// TwinCAT 3 PLC project Untitled1
// ProgramVersion: 3.1.4023.0
// libraries:
//   CmpBitmapPool, * (System)
//   Tc2_MC2, * (Beckhoff Automation GmbH)
//   Tc2_Standard, * (Beckhoff Automation GmbH)
//   Tc2_System, * (Beckhoff Automation GmbH)
//   Tc2_Utilities, * (Beckhoff Automation GmbH)
//   Tc3_Module, * (Beckhoff Automation GmbH)
//   Tc3_PackML_V2, * (Beckhoff Automation GmbH)
// project tree:
//   DUTs/ A21ToolStorage.TcDUT (not stored), Bundle.TcDUT (not stored), Interval.TcDUT (not stored), PositionMaterials.TcDUT (not stored)
//   DUTs/Alarms and Status/ A21Alarms.TcPOU, PMLStackLight.TcPOU (not stored)
//   DUTs/Enums/ A21.TcDUT (not stored), Chipboard.TcDUT (not stored), ConveyorMode.TcDUT (not stored), SectionEnum.TcDUT (not stored), Surface.TcDUT (not stored), WoodBunk.TcDUT (not stored)
//   DUTs/Insertion Package/Drives/ AirPiston.TcPOU (not stored), ClearLinkMC.TcPOU, SimplePiston.TcPOU
//   DUTs/Insertion Package/ Homing.TcDUT (not stored), Insertion.TcPOU, SuctionPad.TcDUT (not stored)
//   DUTs/Insertion Package/Prototypes/ FBA_Drive.TcPOU (not stored), FBA_TrifectaDrive.TcPOU, I_ContinuousDrive.TcIO (not stored), I_Drive.TcIO (not stored), I_EncodedDrive.TcIO (not stored), I_PositionalDrive.TcIO
//   DUTs/Machines/ Conveyor.TcPOU, ConveyorLL.TcPOU, EOAT.TcDUT (not stored), KukaRobot.TcPOU (not stored), RobotA21.TcPOU (not stored), StrapMachine.TcPOU (not stored)
//   DUTs/Material Holders/ MaterialHolder.TcPOU (not stored), MaterialSlot.TcDUT (not stored), SkidMagazine.TcPOU (not stored), StagingTable.TcPOU (not stored)
//   GVLs/ ContainerArrays.TcGVL (not stored), GVL.TcGVL (not stored), Hardware.TcGVL, Misc.TcGVL (not stored)
//   / PlcTask.TcTTO (not stored)
//   POUs/A21a - Chipboard/AOIs/ AOI_LoadChipboard.TcPOU (not stored)
//   POUs/A21b - Wood Bunk/AOIs/ AOI_LoadWoodBunk.TcPOU, AOI_StageWoodBunk.TcPOU (not stored), AOI_StagingTemplate.TcPOU
//   POUs/ CallHardware.TcPOU, FB_System.TcPOU, MAIN.TcPOU
//   POUs/Hardware Functions/ InsertionQuality.TcPOU (not stored), SetSuctionsPtrArr.TcPOU (not stored), SuctionQuality.TcPOU (not stored), SuctionQualityPtrArr.TcPOU (not stored), SetSuctions.TcPOU (not stored), SetupHardware.TcPOU (not stored)
//   POUs/A21a - Chipboard/ ChipboardEx.TcPOU
//   POUs/A21b - Wood Bunk/ WoodBunkEx.TcPOU
//   POUs/Utility/ AddToArray.TcPOU, AddToStringArray.TcPOU (not stored), ArrayIsEmpty.TcPOU, CleanStringsArray.TcPOU (not stored), IntegerBitAccess.TcPOU (not stored), IntegerToBoolArray.TcPOU (not stored), JoinStrings.TcPOU (not stored), WithinTolerance.TcPOU (not stored)
// real-time tasks:
//   TASK PlcTask: cycle T#10ms, priority 20, ADS port 350
// I/O:
//   DEVICE Device 1 (EtherCAT) (disabled), AmsNetId 192.168.101.188.2.1
//     EK1200 [EK1200-5000 EtherCAT Power supply (2A E-Bus)]
//       IPC_O [EL2809 16Ch. Dig. Output 24V, 0.5A]
//       JUNC_A21 [EK1122 2 port EtherCAT junction]
//         A21_C4 [EK1100 EtherCAT Coupler (2A E-Bus)]
//           A21_C4_I1 [EL1809 16Ch. Dig. Input 24V, 3ms]
//           A21_C4_O2 [EL2809 16Ch. Dig. Output 24V, 0.5A]
//           A21_C4_O3 [EL2809 16Ch. Dig. Output 24V, 0.5A]
//           BRIDGE_ROBOT1 [EL6695 EtherCAT Bridge terminal (Primary)]
//           A21_C4_END [EL9011 End Terminal]
//         A21_SB01 [EP1809-0021 16 Ch. Dig. Input 24V, 3ms, M8]
//         A21_SB05 [EP1008-0001 8 Ch. Dig. Input 24V, 3ms, M8]
//         A21_SB04 [EP1809-0021 16 Ch. Dig. Input 24V, 3ms, M8]
//         A21_SB03 [EP1008-0001 8 Ch. Dig. Input 24V, 3ms, M8]
//         A21_C1 [EK1100 EtherCAT Coupler (2A E-Bus)]
//           A21_C1_I1 [EL1809 16Ch. Dig. Input 24V, 3ms]
//           A21_C1_O2 [EL2809 16Ch. Dig. Output 24V, 0.5A]
//           BRIDGE_ROBOT2 [EL6695 EtherCAT Bridge terminal (Primary)]
//           A21_C1_END [EL9011 End Terminal]
//         A21_SB02 [EP1809-0021 16 Ch. Dig. Input 24V, 3ms, M8]
//         A21_SB07 [EP1008-0001 8 Ch. Dig. Input 24V, 3ms, M8]
//         A21_SB06 [EP1008-0001 8 Ch. Dig. Input 24V, 3ms, M8]
//   DEVICE Device 2 (TC3 EIP Scanner) (disabled), AmsNetId 192.168.101.188.3.1
//     ClearLink // <INFO> 169.254.0.152, ClearLink (ProdCode: 1, Rev: 2.93, Mac: 24:15:10:b0:30:37) </INFO> <EDS> C:\TwinCAT\3.1\Config\Io\EtherNetIP\clearlink_2.92.eds </EDS>
// variable links:
//   Untitled1/Untitled1 Instance <-> Device 1 (EtherCAT)/EK1200/JUNC_A21/A21_C1/A21_C1_I1
//     PlcTask Inputs/Hardware.strapperA21.atBundleLevel <-> Channel 6/Input
//     PlcTask Inputs/Hardware.strapperA21.done <-> Channel 4/Input
//     PlcTask Inputs/Hardware.strapperA21.error <-> Channel 1/Input
//     PlcTask Inputs/Hardware.strapperA21.home <-> Channel 5/Input
//     PlcTask Inputs/Hardware.strapperA21.ready <-> Channel 2/Input
//   Untitled1/Untitled1 Instance <-> Device 1 (EtherCAT)/EK1200/JUNC_A21/A21_C1/A21_C1_O2
//     PlcTask Outputs/Hardware.strapperA21.enable <-> Channel 2/Output
//     PlcTask Outputs/Hardware.strapperA21.execute <-> Channel 1/Output
//     PlcTask Outputs/Hardware.strapperA21.reset <-> Channel 3/Output
//   Untitled1/Untitled1 Instance <-> Device 1 (EtherCAT)/EK1200/JUNC_A21/A21_C1/BRIDGE_ROBOT2
//     PlcTask Inputs/Hardware.robot2.inputs[{2..20}] <-> IO Inputs/In_{2..20}  (19 links)
//     PlcTask Inputs/Hardware.robot2.inputs[1] <-> IO Inputs/In
//     PlcTask Inputs/Hardware.robot2.offline <-> SYNC Inputs/External device not connected
//     PlcTask Outputs/Hardware.robot2.outputs[{2..20}] <-> IO Outputs/Out_{2..20}  (19 links)
//     PlcTask Outputs/Hardware.robot2.outputs[1] <-> IO Outputs/Out
//   Untitled1/Untitled1 Instance <-> Device 1 (EtherCAT)/EK1200/JUNC_A21/A21_C4/A21_C4_I1
//     PlcTask Inputs/Hardware.suctionA21Top[1].occupied <-> Channel 9/Input
//     PlcTask Inputs/Hardware.suctionA21Top[2].occupied <-> Channel 10/Input
//     PlcTask Inputs/Hardware.suctionA21Top[3].occupied <-> Channel 11/Input
//     PlcTask Inputs/Hardware.verticalDriveA21Left.home <-> Channel 3/Input
//     PlcTask Inputs/Hardware.verticalDriveA21Left.innerLimit <-> Channel 1/Input
//     PlcTask Inputs/Hardware.verticalDriveA21Left.outerLimit <-> Channel 2/Input
//     PlcTask Inputs/Hardware.verticalDriveA21Right.home <-> Channel 7/Input
//     PlcTask Inputs/Hardware.verticalDriveA21Right.innerLimit <-> Channel 5/Input
//     PlcTask Inputs/Hardware.verticalDriveA21Right.outerLimit <-> Channel 6/Input
//   Untitled1/Untitled1 Instance <-> Device 1 (EtherCAT)/EK1200/JUNC_A21/A21_C4/A21_C4_O2
//     PlcTask Outputs/Hardware.horizontalDriveA21Left.valveExtend <-> Channel 5/Output
//     PlcTask Outputs/Hardware.horizontalDriveA21Left.valveRetract <-> Channel 6/Output
//     PlcTask Outputs/Hardware.horizontalDriveA21Right.valveExtend <-> Channel 15/Output
//     PlcTask Outputs/Hardware.horizontalDriveA21Right.valveRetract <-> Channel 16/Output
//     PlcTask Outputs/Hardware.suctionA21Left[{1..4}].enable <-> Channel {7..10}/Output  (4 links)
//     PlcTask Outputs/Hardware.verticalDriveA21Left.brakeRelease <-> Channel 4/Output
//     PlcTask Outputs/Hardware.verticalDriveA21Right.brakeRelease <-> Channel 14/Output
//   Untitled1/Untitled1 Instance <-> Device 1 (EtherCAT)/EK1200/JUNC_A21/A21_C4/A21_C4_O3
//     PlcTask Outputs/Hardware.pistonA21Bottom.pistonExtend <-> Channel 5/Output
//     PlcTask Outputs/Hardware.pistonA21Bottom.pistonRetract <-> Channel 6/Output
//     PlcTask Outputs/Hardware.suctionA21Bottom[1].enable <-> Channel 7/Output
//     PlcTask Outputs/Hardware.suctionA21Bottom[2].enable <-> Channel 8/Output
//     PlcTask Outputs/Hardware.suctionA21Right[{1..4}].enable <-> Channel {1..4}/Output  (4 links)
//     PlcTask Outputs/Hardware.suctionA21Top[1].enable <-> Channel 9/Output
//     PlcTask Outputs/Hardware.suctionA21Top[2].enable <-> Channel 10/Output
//     PlcTask Outputs/Hardware.suctionA21Top[3].enable <-> Channel 11/Output
//   Untitled1/Untitled1 Instance <-> Device 1 (EtherCAT)/EK1200/JUNC_A21/A21_C4/BRIDGE_ROBOT1
//     PlcTask Inputs/Hardware.robot1.inputs[{2..20}] <-> IO Inputs/In_{2..20}  (19 links)
//     PlcTask Inputs/Hardware.robot1.inputs[1] <-> IO Inputs/In
//     PlcTask Inputs/Hardware.robot1.offline <-> SYNC Inputs/External device not connected
//     PlcTask Outputs/Hardware.robot1.outputs[{2..20}] <-> IO Outputs/Out_{2..20}  (19 links)
//     PlcTask Outputs/Hardware.robot1.outputs[1] <-> IO Outputs/Out
//   Untitled1/Untitled1 Instance <-> Device 1 (EtherCAT)/EK1200/JUNC_A21/A21_SB01
//     PlcTask Inputs/ContainerArrays.tableHmiA21Left[{1..10}].occupied <-> Channel {1..10}/Input  (10 links)
//     PlcTask Inputs/Hardware.horizontalDriveA21Left.home <-> Channel 11/Input
//     PlcTask Inputs/Hardware.insertionA21Left.contact <-> Channel 12/Input
//     PlcTask Inputs/Hardware.suctionA21Left[{1..4}].occupied <-> Channel {13..16}/Input  (4 links)
//   Untitled1/Untitled1 Instance <-> Device 1 (EtherCAT)/EK1200/JUNC_A21/A21_SB02
//     PlcTask Inputs/ContainerArrays.tableHmiA21Right[{1..10}].occupied <-> Channel {1..10}/Input  (10 links)
//     PlcTask Inputs/Hardware.horizontalDriveA21Right.home <-> Channel 11/Input
//     PlcTask Inputs/Hardware.insertionA21Right.contact <-> Channel 12/Input
//     PlcTask Inputs/Hardware.suctionA21Right[{1..4}].occupied <-> Channel {13..16}/Input  (4 links)
//   Untitled1/Untitled1 Instance <-> Device 1 (EtherCAT)/EK1200/JUNC_A21/A21_SB07
//     PlcTask Inputs/Hardware.pistonA21Bottom.extended <-> Channel 5/Input
//     PlcTask Inputs/Hardware.pistonA21Bottom.retracted <-> Channel 4/Input
//     PlcTask Inputs/Hardware.suctionA21Bottom[1].occupied <-> Channel 6/Input
//     PlcTask Inputs/Hardware.suctionA21Bottom[2].occupied <-> Channel 7/Input
//   Untitled1/Untitled1 Instance <-> Device 2 (TC3 EIP Scanner)/ClearLink
//     PlcTask Inputs/Hardware.verticalDriveA21Left.hlfb <-> Connection 1 (Input/Output)/Inputs/Motor0 HLFB Duty
//     PlcTask Inputs/Hardware.verticalDriveA21Right.hlfb <-> Connection 1 (Input/Output)/Inputs/Motor1 HLFB Duty
//     PlcTask Outputs/Hardware.verticalDriveA21Left.outputRegister <-> Connection 1 (Input/Output)/Outputs/Motor0 Out Reg
//     PlcTask Outputs/Hardware.verticalDriveA21Left.pulse <-> Connection 1 (Input/Output)/Outputs/Motor0 Trig Pulses
//     PlcTask Outputs/Hardware.verticalDriveA21Right.outputRegister <-> Connection 1 (Input/Output)/Outputs/Motor1 Out Reg
//     PlcTask Outputs/Hardware.verticalDriveA21Right.pulse <-> Connection 1 (Input/Output)/Outputs/Motor1 Trig Pulses

// ---- GVLs/Hardware.TcGVL
//{attribute 'qualified_only'}
VAR_GLOBAL
	robot1 : RobotA21;
	robot2 : RobotA21;
	
	toolStorageA21Left : A21ToolStorage;
	toolStorageA21Right : A21ToolStorage;
	
	skidA21Left : SkidMagazine;
	skidA21Right : SkidMagazine;
	
	magazineA21Left : SkidMagazine;
	magazineA21Right : SkidMagazine;
	stagingTableLeft : StagingTable;
	stagingTableRight : StagingTable;
	
	strapperA21 : StrapMachine;
	
	horizontalDriveA21Left, horizontalDriveA21Right : AirPiston := (
		limitSensorDefaultState := FALSE,
		useBrake := FALSE);
	
	verticalDriveA21Left, verticalDriveA21Right : ClearLinkMC := (
		limitSensorDefaultState := TRUE, 
		homingDirectionOut := TRUE, //outwards (up)
		minPosition := 0,
		displacementPerRotation := 1,
		unitsPerPulse := 8000); //0.1x gearbox, 10 revs/pulse to compensate
		
	insertionA21Left, insertionA21Right : Insertion;
	
	pistonA21Bottom : SimplePiston;
	
	suctionA21Top : ARRAY[1..3] OF SuctionPad;
	suctionA21Left : ARRAY[1..4] OF SuctionPad;
	suctionA21Right : ARRAY[1..4] OF SuctionPad; 
	suctionA21Bottom : ARRAY[1..2] OF SuctionPad;
	
	stackLightA21 : PMLStackLight;
	alarmsA21 : A21Alarms;
END_VAR

// ---- DUTs/Insertion Package/Prototypes/I_PositionalDrive.TcIO
INTERFACE I_PositionalDrive EXTENDS I_Drive

PROPERTY CurrentPosition : LREAL
GET
END_GET
SET
END_SET
END_PROPERTY

METHOD ABSTRACT moveAbsolute : BOOL
VAR_INPUT
	newTarget : LREAL; 
END_VAR
END_METHOD

METHOD ABSTRACT moveRelative : BOOL
VAR_INPUT
	distance : LREAL;
END_VAR
END_METHOD

PROPERTY TargetPosition : LREAL
GET
END_GET
SET
END_SET
END_PROPERTY

END_INTERFACE

// ---- DUTs/Insertion Package/Drives/ClearLinkMC.TcPOU
FUNCTION_BLOCK ClearLinkMC EXTENDS FBA_TrifectaDrive IMPLEMENTS I_EncodedDrive
VAR_OUTPUT
	pulse AT %Q* : INT;
	brakeRelease AT %Q* : BOOL := TRUE;
	enable : BOOL;
	A : BOOL;
	B : BOOL;
	clear : BOOL;
END_VAR
VAR	
	hlfb AT %I* : REAL := -9999; //high level feedback, if -9999 then servo is idle
	
	outputRegister AT %Q* : INT;
	pulseRequest : INT;
	
	homingDelay : TON;
	resetPulse : TP;
	
	mode : (HOLD, TARGET, CONTINUOUS, RESET_ERR);
	calculation : (IDLE, DOWN, UP, CALCULATE, DONE);
	maxPosition : LREAL;
	
	position, targetPos : LREAL;
	
	pulsePosition : INT;
	pulseCounter : INT;
	rotationsPerPulse : INT; //revolutions per pulse
	displacementPerPulse : LREAL; //displacement per pulse
END_VAR
VAR_STAT CONSTANT
	resetWidth : TIME := T#500MS;
	delayWidth : TIME := T#500MS;
END_VAR
VAR //constructor
	homingDirectionOut : BOOL; 			//homing direction - see <A>
	minPosition : LREAL;
	displacementPerRotation : LREAL; 	//displacement per revolution	
	unitsPerPulse : INT := 800; 		//800 Teknic units per rotation - default setting is 800 units (1 rotation) per pulse
END_VAR

//M-connector output register
outputRegister.0 := enable AND bEnable; 	//enable
outputRegister.1 := A; 						//direction bit - T = outwards, F = inwards
outputRegister.2 := B; 						//homing bit - after startup, set to TRUE to begin homing, then set to FALSE to finish homing
outputRegister.3 := clear; 					//reset bit

rotationsPerPulse := unitsPerPulse/800; //Teknic constant - 800 units per rotation
displacementPerPulse := displacementPerRotation * rotationsPerPulse;

resetPulse(IN:= , PT:= resetWidth, Q=> clear, ET=> ); //reset pulse

IF NOT enable AND NOT AtInnerLimit THEN
	homingComplete := FALSE;
	step := Homing.IDLE;
	mode := HOLD;
END_IF

override();

CASE mode OF		
	HOLD: //hold current position, no motion
		pulse := 0;
		pulseRequest := 0;
	
	TARGET:	//target a given position
		
		IF WithinTolerance(position, targetPos, displacementPerPulse) THEN
			pulseRequest := 0;
			pulse := 0;
			mode := HOLD;
			
		ELSIF NOT Active THEN
			A :=  position < targetPos;
			(*
			2 options to traverse to a target position:
				a)  send all pulses at once - continuous motion but may exceed limits, check for bounds before setting
				b)  1 pulse at a time - choppy but safer
			*)
			targetPos := MAX(targetPos, minPosition); //if below minPosition, set to minPosition
			targetPos := MIN(targetPos, maxPosition); //if above maxPosition, set to maxPosition
			
			pulseRequest := TO_INT(ABS(position - targetPos)/displacementPerPulse);
			//pulseRequest := 1;
		END_IF
		
	CONTINUOUS: //single pulses in the direction specified by moveContinuous()
		pulseRequest := 1;
		
	RESET_ERR: //reset pulse, servo may need to be rehomed aftewards
		pulse := 0;
		pulseRequest := 0;
		resetPulse.IN := TRUE;
		
		IF resetPulse.Q THEN
			resetPulse.IN := FALSE;
			mode := HOLD;
		END_IF
		
END_CASE

sequence();

PROPERTY Active : BOOL
GET
Active := hlfb <> -9999;
END_GET
END_PROPERTY

{attribute 'monitoring':='call'}
PROPERTY AtOuterLimit : BOOL
GET
AtOuterLimit := outerLimit <> limitSensorDefaultState;
END_GET
END_PROPERTY

METHOD PRIVATE calculatePositions : BOOL
(*
the purpose of this method is calculate the position at the outer limit

complete a full range traverse while counting the pulses, then multiply
	displacement per rotation
	rotations per pulse
	number of pulses for the traversal
and add to position at inner limit to get position at outer limit
*)
CASE calculation OF
	IDLE:
		calculation := DOWN;
		
	DOWN:
		moveContinuous(direction := MC_Negative_Direction);
		IF AtInnerLimit THEN
			calculation := UP;
			pulseCounter := 0;
		END_IF
		
	UP:
		moveContinuous(direction := MC_Positive_Direction);
		IF AtHome THEN
			maxPosition := minPosition + (displacementPerRotation * rotationsPerPulse * pulseCounter);
			calculation := DONE;
		END_IF
		
	DONE:
		calculation := 0;
		calculatePositions := TRUE;
		
END_CASE
END_METHOD

PROPERTY CurrentPosition : LREAL
GET
CurrentPosition := position;

//CurrentPosition := pulsePosition * displacementPerPulse;
END_GET
SET
position := CurrentPosition;
END_SET
END_PROPERTY

PROPERTY Error : BOOL
GET
END_GET
END_PROPERTY

METHOD homingSequence : BOOL
homingDelay(IN:= , PT:= delayWidth, Q=> , ET=> );

CASE step OF
	Homing.IDLE:
		enable := TRUE;
		A := FALSE;
		B := TRUE;
		brakeRelease := TRUE;
		
		homingComplete := FALSE;
		
		homingDelay.IN := TRUE;
		IF homingDelay.Q THEN
			homingDelay.IN := FALSE;
			//step := Homing.START;
			step := Homing.RETRY;
		END_IF
		
	Homing.START:
		IF homingDelay.Q THEN
			homingDelay.IN := FALSE;
			step := Homing.SET;
			
		ELSIF AtHome THEN
			homingDelay.IN := TRUE;
			
		ELSIF AtOuterLimit THEN
			step := Homing.RETRY;
		
		ELSE
			enable := TRUE;
			A := FALSE;
			B := TRUE;
			brakeRelease := TRUE;
		
		END_IF
	
	Homing.RETRY:
		IF AtInnerLimit THEN
			homingDelay.IN := TRUE;
			enable := FALSE;
			
			IF homingDelay.Q THEN
				homingDelay.IN := FALSE;
				step := Homing.START;
			END_IF
			
		ELSE
			enable := TRUE;
			A := FALSE;
			B := FALSE;
			brakeRelease := TRUE;
			
			mode := CONTINUOUS;
		END_IF

	Homing.SET:
		enable := TRUE;
		A := FALSE;
		B := FALSE;
		brakeRelease := TRUE;
		
		IF calculatePositions() THEN
			step := Homing.DONE;
		END_IF
		
	Homing.DONE:
		homingSequence := homingComplete := TRUE;
		
		pulsePosition := 0;
		
		mode := HOLD;
		step := Homing.IDLE;
	
END_CASE
END_METHOD

{attribute 'TcRpcEnable'}
METHOD moveAbsolute : BOOL
VAR_INPUT
	newTarget : LREAL;
END_VAR
IF target >= maxPosition AND target <= minPosition THEN
	A :=  position < targetPos;
	targetPos := newTarget;
	mode := TARGET;
	
	moveAbsolute := TRUE;
END_IF
END_METHOD

{attribute 'TcRpcEnable'}
METHOD moveContinuous : BOOL
VAR_INPUT
	direction : MC_Direction;
END_VAR
IF direction = MC_Negative_Direction THEN
	A := FALSE;
ELSIF direction = MC_Positive_Direction THEN
	A := TRUE;
END_IF

mode := CONTINUOUS;
END_METHOD

{attribute 'TcRpcEnable'}
METHOD moveRelative : BOOL
VAR_INPUT
	distance : LREAL;
END_VAR
targetPos := targetPos + distance;

mode := TARGET;
END_METHOD

METHOD PRIVATE override : BOOL
VAR_INPUT
END_VAR
(*
allowable motion is between AtHome and AtInnerLimit
*)
IF AtHome AND NOT Active THEN
	IF homingDirectionOut THEN //homing is outwards
		position := maxPosition;
		pulsePosition := pulseCounter;
	ELSE
		position := minPosition;
		pulsePosition := 0;
	END_IF
	

ELSIF AtInnerLimit AND NOT Active THEN
	IF homingDirectionOut THEN //homing is outwards
		position := minPosition;
		pulsePosition := 0;
	ELSE
		position := maxPosition;
		pulsePosition := pulseCounter;
	END_IF
END_IF

CASE mode OF		
	HOLD:
		//
	
	TARGET:
		IF
			(AtHome AND TargetPosition > CurrentPosition) OR
			(AtInnerLimit AND TargetPosition > CurrentPosition) OR
			(AtOuterLimit AND TargetPosition < CurrentPosition)
		THEN
			mode := HOLD;
		END_IF
		
	CONTINUOUS:
		IF
			(AtHome AND A) OR
			(AtInnerLimit AND A) OR
			(AtOuterLimit AND NOT A)
		THEN
			mode := HOLD;
		END_IF
		
	RESET_ERR:
		//
		
END_CASE
END_METHOD

METHOD reset : BOOL
VAR_INPUT
END_VAR
mode := RESET_ERR;
END_METHOD

METHOD PRIVATE sequence : BOOL
VAR_INPUT
END_VAR
IF Active THEN //servo is active
	IF A THEN //positive direction
		position := position + (displacementPerPulse * pulse);
		pulsePosition := pulsePosition + pulse;
		
		pulseCounter := pulseCounter + pulse;
	ELSE //negative direction
		position := position - (displacementPerPulse * pulse);
		pulsePosition := pulsePosition - pulse;
		
		pulseCounter := pulseCounter - pulse;
	END_IF
	pulse := 0; //pulses already received, can be set to 0 so position change is not compounded

ELSIF pulse = 0 THEN //servo is not active
	pulse := pulseRequest;
END_IF

pulseRequest := 0; //remove this if not working as intended
END_METHOD

METHOD stop : BOOL
VAR_INPUT
END_VAR
mode := HOLD;
END_METHOD

PROPERTY TargetPosition : LREAL
GET
END_GET
SET
targetPos := TargetPosition;
END_SET
END_PROPERTY

METHOD toHome : BOOL
VAR_INPUT
END_VAR
IF homingDirectionOut THEN
	moveAbsolute(newTarget := maxPosition);
ELSE
	moveAbsolute(newTarget := minPosition);
END_IF
END_METHOD

END_FUNCTION_BLOCK

// ---- DUTs/Insertion Package/Prototypes/FBA_TrifectaDrive.TcPOU
FUNCTION_BLOCK ABSTRACT FBA_TrifectaDrive EXTENDS FBA_Drive
VAR
	outerLimit AT %I* : BOOL;
END_VAR
(*
this abstract FB adds a rear limit sensor to FBA_Drive
*)

{attribute 'monitoring':='call'}
PROPERTY AtOuterLimit : BOOL
GET
AtOuterLimit := outerLimit <> limitSensorDefaultState;
END_GET
END_PROPERTY

END_FUNCTION_BLOCK

// ---- DUTs/Insertion Package/Insertion.TcPOU
FUNCTION_BLOCK Insertion //2d insertion that combines a slider (alignment) and screw (push)
VAR_INPUT
	enable : BOOL;
END_VAR
VAR_INPUT //interface references to existing drives
	slider : I_EncodedDrive;
	screw : I_ContinuousDrive;
END_VAR
VAR_OUTPUT
	contact AT %I* : BOOL;
	
	active : BOOL;
	error : BOOL;
	home : BOOL;
	
	homingComplete : BOOL;
	
	sliderPos : LREAL;
END_VAR
(*
this FB encapsulates 2 drives into a generic insertion machine
both drives should be declared externally in Hardware GVL as a concrete FB
Insertion instance should be declared and called in module scope, with the drives from Hardware GVL passed in by Interface reference
*)

homingComplete := slider.HomeSet AND screw.HomeSet;

active := slider.Active OR screw.Active;
error := slider.Error OR screw.Error;
home := slider.AtHome AND screw.AtHome;

sliderPos := slider.CurrentPosition;

METHOD align : BOOL
VAR_INPUT
	targetPos : REAL;
END_VAR
slider.moveAbsolute(newTarget := targetPos);
END_METHOD

METHOD homingSequence : BOOL
VAR_INPUT
END_VAR
IF NOT slider.homeSet THEN
	slider.homingSequence();
END_IF

IF NOT screw.homeSet THEN
	screw.homingSequence();
END_IF

homingSequence := homingComplete;
END_METHOD

METHOD press : BOOL
VAR_INPUT
END_VAR
screw.moveContinuous(direction := MC_Negative_Direction);
END_METHOD

METHOD release : BOOL
VAR_INPUT
END_VAR
screw.moveContinuous(direction := MC_Positive_Direction);
END_METHOD

METHOD reset : BOOL
VAR_INPUT
END_VAR
slider.reset();
screw.reset();
END_METHOD

METHOD stop : BOOL
VAR_INPUT
END_VAR
screw.stop();
slider.stop();
END_METHOD

METHOD toHome : BOOL
VAR_INPUT
END_VAR
slider.toHome();
screw.toHome();

toHome := slider.AtHome AND screw.AtHome;
END_METHOD

METHOD traverse : BOOL
VAR_INPUT
	direction : MC_Direction;
END_VAR
slider.moveContinuous(direction := MC_Negative_Direction);
END_METHOD

END_FUNCTION_BLOCK

// ---- DUTs/Insertion Package/Drives/SimplePiston.TcPOU
FUNCTION_BLOCK SimplePiston
VAR_INPUT
	bEnable : BOOL;
END_VAR
VAR_OUTPUT
	pistonExtend AT %Q* : BOOL;
	pistonRetract AT %Q* : BOOL;
	
	extended AT %I* : BOOL;
	retracted AT %I* : BOOL;
	
	busy : BOOL;
END_VAR
VAR
	mode : (HOLD, IN, OUT);
END_VAR

IF
	NOT bEnable OR
	(retracted AND_THEN (pistonRetract OR mode = OUT)) OR
	(extended AND_THEN (pistonExtend OR mode = IN))
THEN
	mode := HOLD;
END_IF

CASE mode OF
	HOLD:
		pistonRetract := FALSE;
		pistonExtend := FALSE;
		
	IN:
		pistonRetract := FALSE;
		pistonExtend := TRUE;
	
	OUT:
		pistonRetract := TRUE;
		pistonExtend := FALSE;
	
END_CASE

busy := mode = IN OR mode = OUT;

METHOD extend : BOOL
VAR_INPUT
END_VAR
mode := IN;
END_METHOD

METHOD retract : BOOL
VAR_INPUT
END_VAR
mode := OUT;

retract := retracted;
END_METHOD

METHOD stop : BOOL
VAR_INPUT
END_VAR
pistonExtend := FALSE;
pistonRetract := FALSE;
mode := HOLD;
END_METHOD

END_FUNCTION_BLOCK

// ---- DUTs/Alarms and Status/A21Alarms.TcPOU
FUNCTION_BLOCK A21Alarms
VAR_OUTPUT
	panelPowerOn : BOOL;
	safetyOk : BOOL;
	airPressureOk : BOOL;
END_VAR
VAR_OUTPUT
	alarm : BOOL;
END_VAR

alarm :=
	NOT panelPowerOn OR 
	NOT safetyOk OR
	NOT airPressureOk;

END_FUNCTION_BLOCK

// ---- DUTs/Machines/Conveyor.TcPOU
FUNCTION_BLOCK Conveyor
VAR
	enable AT %Q* : BOOL := TRUE;
	direction AT %Q* : BOOL; //FALSE = forward, TRUE = backward
	pulse AT %Q* : BOOL;
	reset AT %Q* : BOOL;
	
	sensorEntry AT %I* : BOOL;
	sensorExit AT %I* : BOOL;

	lifterEnable AT %Q* : BOOL := TRUE;
	lifterDirection AT %Q* : BOOL; //FALSE = up, TRUE = down
	lifterPulse AT %Q* : BOOL;
	lifterReset AT %Q* : BOOL;
END_VAR
VAR_OUTPUT
	operation : ConveyorMode;
	request : ConveyorMode;
	
	error AT %I* : BOOL;
	lifterError AT %I* : BOOL;
	
	position AT %I* : REAL;
	velocity AT %I* : REAL;
	
	hasLifter : BOOL;
	extended AT %I* : BOOL;
	retracted AT %I* : BOOL;
END_VAR
VAR
	lifterMode : (HOLD, UP, DOWN); 
	lifterMode2 : (LIFTER_EXTEND, LIFTER_RETRACT);
	
	//pulses are assumed to be low-high-low
	pulser : TP;
	lifterPulser : TP;
END_VAR
VAR_STAT CONSTANT
	pulseWidth : TIME := T#25MS;
END_VAR
(*
this version of Conveyor is to be implemented as a linked list,
	allowing it to control its own mode internally -
	without the use of an external conveyor control module - 
	eliminating the ability for other modules to modify its mode
*)

lifterPulser(IN:= , PT:= pulseWidth, Q=> lifterPulse, ET=> );
lifterPulser.IN := 
	hasLifter AND
	lifterEnable AND 
	NOT lifterError AND 
	NOT lifterReset AND 
	( (lifterMode = LIFTER_EXTEND AND NOT extended) OR (lifterMode = LIFTER_RETRACT AND NOT retracted) ) AND
	lifterPulser.Q; //self-ending pulse

override();

CASE lifterMode OF
	HOLD:
		lifterDirection := TRUE;
		lifterPulse := FALSE;
		
	UP:
		lifterDirection := FALSE;
		lifterPulse := NOT lifterPulse;
	
	DOWN:
		lifterDirection := TRUE;
		lifterPulse := NOT lifterPulse;
	
END_CASE

//conveyors do not move independently like motion drives, their operation is set by an additional conveyor control module
traverseSequence();

METHOD backward : BOOL
VAR_INPUT
END_VAR
END_METHOD

METHOD extend : BOOL
VAR_INPUT
END_VAR
VAR
	noLifter : BOOL;
END_VAR
IF hasLifter THEN
	lifterMode := UP;
	extend := TRUE;
ELSE
	noLifter := TRUE;
END_IF
END_METHOD

METHOD forward : BOOL
VAR_INPUT
END_VAR
END_METHOD

METHOD occupied : BOOL
occupied := sensorExit OR sensorEntry;
END_METHOD

METHOD PRIVATE override : BOOL
VAR_INPUT
END_VAR
IF
	(extended AND lifterMode = UP) OR
	(retracted AND lifterMode = DOWN)
THEN
	lifterMode := HOLD;
END_IF
END_METHOD

METHOD reset : BOOL
VAR_INPUT
END_VAR
position := 0;
velocity := velocity; //no change

extend();
END_METHOD

METHOD retract : BOOL
VAR_INPUT
END_VAR
VAR
	noLifter : BOOL;
END_VAR
IF hasLifter THEN
	lifterMode := DOWN;
	retract := TRUE;
ELSE
	noLifter := TRUE;
END_IF
END_METHOD

METHOD setOperation : BOOL
VAR_INPUT
	newOperation : ConveyorMode;
END_VAR
operation := newOperation;
END_METHOD

METHOD setRequest : BOOL
VAR_INPUT
	requestedMode : ConveyorMode;
END_VAR
request := requestedMode;
END_METHOD

METHOD target : BOOL
VAR_INPUT
	targetPosition : REAL;
END_VAR
END_METHOD

METHOD PRIVATE traverseSequence : BOOL
VAR_INPUT
END_VAR
direction := (operation = ConveyorMode.BACKWARD);

pulser(IN:= , PT:= pulseWidth, Q=> pulse, ET=> );
pulser.IN := 
	enable AND 
	NOT error AND 
	NOT reset AND 
	(operation = ConveyorMode.FORWARD OR operation = ConveyorMode.BACKWARD)
	AND pulser.Q; //ends pulse itself
END_METHOD

END_FUNCTION_BLOCK

// ---- DUTs/Machines/ConveyorLL.TcPOU
FUNCTION_BLOCK ConveyorLL
VAR
	enable AT %Q* : BOOL := TRUE;
	direction AT %Q* : BOOL; //FALSE = forward, TRUE = backward
	pulse AT %Q* : BOOL;
	reset AT %Q* : BOOL;
	
	sensorEntry AT %I* : BOOL;
	sensorExit AT %I* : BOOL;

	lifterEnable AT %Q* : BOOL := TRUE;
	lifterDirection AT %Q* : BOOL; //FALSE = up, TRUE = down
	lifterPulse AT %Q* : BOOL;
	lifterReset AT %Q* : BOOL;
END_VAR
VAR_OUTPUT
	operation : ConveyorMode;
	request : ConveyorMode;
	
	error AT %I* : BOOL;
	lifterError AT %I* : BOOL;
	
	position AT %I* : REAL;
	velocity AT %I* : REAL;
	
	hasLifter : BOOL;
	extended AT %I* : BOOL;
	retracted AT %I* : BOOL;
END_VAR
VAR
	nextConveyor : POINTER TO Conveyor;
	prevConveyor : POINTER TO Conveyor;
	
	lifterMode : (HOLD, LIFTER_EXTEND, LIFTER_RETRACT); 
	
	//pulses are assumed to be low-high-low
	pulser : TP;
	lifterPulser : TP;
END_VAR
VAR_STAT CONSTANT
	pulseWidth : TIME := T#25MS;
END_VAR

pulser(IN:= , PT:= pulseWidth, Q=> pulse, ET=> );
pulser.IN := 
	enable AND 
	NOT error AND 
	NOT reset AND 
	(operation = ConveyorMode.FORWARD OR operation = ConveyorMode.BACKWARD)
	AND pulser.Q; //ends pulse itself

lifterPulser(IN:= , PT:= pulseWidth, Q=> lifterPulse, ET=> );
lifterPulser.IN := 
	hasLifter AND
	lifterEnable AND 
	NOT lifterError AND 
	NOT lifterReset AND 
	( (lifterMode = LIFTER_EXTEND AND NOT extended) OR (lifterMode = LIFTER_RETRACT AND NOT retracted) ) AND
	lifterPulser.Q; //self-ending pulse

override();

CASE lifterMode OF
	HOLD:
		lifterDirection := TRUE;
		lifterPulse := FALSE;
		
	LIFTER_EXTEND:
		lifterDirection := FALSE;
		lifterPulse := NOT lifterPulse;
	
	LIFTER_RETRACT:
		lifterDirection := TRUE;
		lifterPulse := NOT lifterPulse;
	
END_CASE

sequence();

METHOD backward : BOOL
VAR_INPUT
END_VAR
END_METHOD

METHOD extend : BOOL
VAR_INPUT
END_VAR
VAR
	noLifter : BOOL;
END_VAR
IF hasLifter THEN
	lifterMode := UP;
	extend := TRUE;
ELSE
	noLifter := TRUE;
END_IF
END_METHOD

METHOD forward : BOOL
VAR_INPUT
END_VAR
END_METHOD

PROPERTY IsOccupied : BOOL
GET
IsOccupied := sensorExit OR sensorEntry;
END_GET
END_PROPERTY

METHOD PRIVATE override : BOOL
VAR_INPUT
END_VAR
IF
	(extended AND lifterMode = UP) OR
	(retracted AND lifterMode = DOWN)
THEN
	lifterMode := HOLD;
END_IF
END_METHOD

METHOD reset : BOOL
VAR_INPUT
END_VAR
position := 0;
velocity := velocity; //no change

extend();
END_METHOD

METHOD retract : BOOL
VAR_INPUT
END_VAR
VAR
	noLifter : BOOL;
END_VAR
IF hasLifter THEN
	lifterMode := DOWN;
	retract := TRUE;
ELSE
	noLifter := TRUE;
END_IF
END_METHOD

METHOD PRIVATE sequence : BOOL
VAR_INPUT
END_VAR
VAR
	nextOp, prevOp : ConveyorMode;
END_VAR
IF nextConveyor <> 0 THEN
	nextOp := nextConveyor^.operation;
END_IF
IF prevConveyor <> 0 THEN
	prevOp := prevConveyor^.operation;
END_IF


IF IsOccupied THEN
	operation := MAX(nextOp, request, prevOp);
ELSE
	operation := ConveyorMode.IDLE;
END_IF


direction := (operation = ConveyorMode.BACKWARD); //set direction bit

IF hasLifter THEN
	
END_IF
END_METHOD

METHOD setOperation : BOOL
VAR_INPUT
	newOperation : ConveyorMode;
END_VAR
operation := newOperation;
END_METHOD

METHOD setRequest : BOOL
VAR_INPUT
	requestedMode : ConveyorMode;
END_VAR
request := requestedMode;
END_METHOD

METHOD target : BOOL
VAR_INPUT
	targetPosition : REAL;
END_VAR
END_METHOD

END_FUNCTION_BLOCK

// ---- POUs/A21b - Wood Bunk/AOIs/AOI_LoadWoodBunk.TcPOU
FUNCTION_BLOCK AOI_LoadWoodBunk
VAR_INPUT
	execute : BOOL;
END_VAR
VAR_IN_OUT CONSTANT
	sectionID : SectionEnum;
END_VAR
VAR_IN_OUT
	robot : RobotA21;
	table : StagingTable;
	//suctions : ARRAY[*] OF SuctionPad;
	//if assigned using . operator instead of (), this becomes a pointer - use numPads isntead of UPPER_BOUND/LOWER_BOUND
	loadedMaterials : ARRAY[*] OF STRING;
END_VAR
VAR_INPUT
	suctions : POINTER TO SuctionPad;
	surfaceID : Surface;
	material : STRING;	
	numPads : DINT;
END_VAR
VAR_OUTPUT
	busy : BOOL;
	done : BOOL;
	error : BOOL;
	
	recovery : BOOL;
	failCounter : INT;
	
	donePulse : BOOL;
END_VAR
VAR
	run : BOOL;
	trigger : R_TRIG;
	doneTrigger : R_TRIG;
	
	slot : INT;
	
	suctionTimer : TON;
	step : (IDLE, PREP_ROBOT, GET_FROM_TABLE, LOAD_TO_INSERTION, COMPLETE, RECOVERY_IDLE, RECOVERY_REMOVE, RECOVERY_STAGE);
END_VAR
VAR
	i : DINT;
	test : BOOL;
	
	iWoodBunk : WoodBunk;
END_VAR
VAR CONSTANT
	suctionDelay : TIME := T#2S;
	suctionDistance : INT := 10;
END_VAR

{warning disable C0371}

trigger(CLK:= execute, Q=> );
doneTrigger(CLK:= done, Q=> donePulse);
busy := trigger.Q OR step > 0;

IF step > IDLE AND_THEN NOT preExecution() THEN //conditions to track before execution
	RETURN;
END_IF

(*
if required bunk was not found on table - restage entire table
if bunk was not loaded correctly - remove bunk, then restage entire table
*)

CASE step OF
	IDLE:
		IF trigger.Q THEN //reset outputs
			done := FALSE;
			error := FALSE;
			recovery := FALSE;
			
			step := PREP_ROBOT;
		END_IF
		
	PREP_ROBOT:
		robot.clearCommand();
		IF robot.Ready THEN
			step := GET_FROM_TABLE;
			slot := 0;
		END_IF
		
	GET_FROM_TABLE:		
		IF slot < 1 AND_THEN NOT table.findSlot(material := material, index => slot) THEN
			step := RECOVERY_STAGE;
			RETURN;
		END_IF
		
		
		
		IF NOT table.isOccupied(i := slot) AND table.getSlot(i := slot) <> '' THEN //move from table to robot gripper
			robot.HoldMaterial := table.getSlot(i := slot);
			table.remove(i := slot, material => );
		END_IF
		
		IF robot.Done THEN
			step := COMPLETE;
			RETURN;
		ELSIF robot.materialAtHoldingPosition >= 1 AND robot.materialAtHoldingPosition <= 8 THEN
			step := LOAD_TO_INSERTION;
			RETURN;
		END_IF
		
		CASE surfaceID OF
			Surface.TOP: 					robot.setGroup(group := 1, value := A21.LOAD_BUNK_TOP); 
			Surface.LEFT, Surface.RIGHT: 	robot.setGroup(group := 1, value := A21.LOAD_BUNK_SIDE);
			Surface.BOTTOM: 				robot.setGroup(group := 1, value := A21.LOAD_BUNK_BOTTOM);
		END_CASE
		robot.setGroup(group := 2, value := slot); 
		
		FOR iWoodBunk:=0 TO WoodBunk.size BY 1 DO
			IF material = TO_STRING(iWoodBunk) THEN
				robot.setGroup(group := 3, value := iWoodBunk);
				EXIT;
			END_IF
		END_FOR
			
	LOAD_TO_INSERTION:
		IF robot.materialAtHoldingPosition > 0 AND robot.HoldMaterial <> '' THEN //move from gripper to insertion
			IF loadedMaterials[surfaceID] = '' THEN //transfer to insertion as is
				loadedMaterials[surfaceID] := robot.HoldMaterial;
			ELSE //join with existing material using underscore _
				loadedMaterials[surfaceID] := JoinStrings(loadedMaterials[surfaceID], robot.HoldMaterial, '_');
			END_IF
			robot.HoldMaterial := '';
		END_IF
		
		CASE surfaceID OF
			Surface.TOP, Surface.BOTTOM:	SetSuctionsPtrArr(suctions := suctions, numPads := numPads, state := TRUE);
			Surface.LEFT, Surface.RIGHT:	SetSuctionsPtrArr(suctions := suctions, numPads := numPads, state := TRUE);
		END_CASE
		
		IF robot.Done THEN
			suctionTimer.IN := FALSE;
			step := COMPLETE;
			RETURN;
		END_IF
		
		suctionTimer(IN:= , PT:= suctionDelay, Q=> , ET=> );
		suctionTimer.IN := TRUE;
		
		IF suctionTimer.Q THEN
			robot.setGroup(group := 9, value := robot.materialAtHoldingPosition);
		END_IF
	
	COMPLETE:
		robot.clearCommand();
		
		//check insertion quality
		IF
			SuctionQualityPtrArr(
				suctions := suctions,
				numPads := numPads,
				insertionMaterial := loadedMaterials[surfaceID],
				recipeMaterial := material)
		THEN
			done := TRUE;
			slot := 0;
			step := 0;
		ELSE //recovery - remove wood bunk and restage
			failCounter := failCounter + 1;
			step := RECOVERY_IDLE;
		END_IF
		
	//---------RECOVERY-----------------------------------------
	RECOVERY_IDLE:
		robot.clearCommand();
		IF robot.Ready THEN
			step := RECOVERY_REMOVE;
		END_IF
		
	RECOVERY_REMOVE:
		IF robot.Done THEN
			step := RECOVERY_STAGE;
			RETURN;
		END_IF
		
		CASE surfaceID OF
			Surface.TOP:					robot.setGroup(group := 1, value := A21.REMOVE_BUNK_TOP);
			Surface.LEFT, Surface.RIGHT:	robot.setGroup(group := 1, value := A21.REMOVE_BUNK_SIDE);
			Surface.BOTTOM:					robot.setGroup(group := 1, value := A21.REMOVE_BUNK_BOTTOM);
		END_CASE
	
	RECOVERY_STAGE:	
		recovery := TRUE;
		error := TRUE;
		
END_CASE

METHOD PRIVATE preExecution : BOOL
VAR_INPUT
END_VAR
{warning disable C0371}
IF material = '' THEN
	done := TRUE;
	RETURN;
END_IF

IF //robot must be ready before execution
	robot.error OR 
	robot.reservation <> sectionID OR 
	robot.tool <> sectionID
THEN
	error := TRUE;
	RETURN;
END_IF

preExecution := TRUE;
END_METHOD

METHOD reset : BOOL
VAR_INPUT
END_VAR
VAR
	temp : AOI_LoadWoodBunk;
END_VAR
//(*
done := FALSE;
error := FALSE;
recovery := FALSE;
slot := 0;
step := 0;

failCounter := 0;
//*)
//THIS^ := temp;
END_METHOD

END_FUNCTION_BLOCK

// ---- POUs/CallHardware.TcPOU
PROGRAM CallHardware

(*
the only purpose of this POU is to call modules from Hardware
may be implemented as a PROGRAM or FUNCTION
may be rewritten in Ladder
*)

robot1();	
robot2();

skidA21Left(slots := skidHmiA21Left);
skidA21Right(slots := skidHmiA21Right);

stagingTableLeft(slots := tableHmiA21Left);
stagingTableRight(slots := tableHmiA21Right);

magazineA21Left(slots := magazineHmiA21Left);
magazineA21Right(slots := magazineHmiA21Right);

strapperA21();

verticalDriveA21Left();
horizontalDriveA21Left();

verticalDriveA21Right();
horizontalDriveA21Right();

pistonA21Bottom();

insertionA21Left(
	enable:= TRUE, 
	slider:= verticalDriveA21Left, 
	screw:= horizontalDriveA21Left, 
	active=> , 
	error=> , 
	home=> , 
	homingComplete=> , 
	sliderPos=> );
	
insertionA21Right(
	enable:= TRUE, 
	slider:= verticalDriveA21Right, 
	screw:= horizontalDriveA21Right, 
	active=> , 
	error=> , 
	home=> , 
	homingComplete=> , 
	sliderPos=> );
	
stackLightA21(
	pmlState:= , 
	lowMaterial:= , 
	materialExhausted:= , 
	red=> , 
	yellow=> , 
	blue=> , 
	green=> );
	
alarmsA21(
	panelPowerOn=> , 
	safetyOk=> , 
	airPressureOk=> , 
	alarm=> );

END_PROGRAM

// ---- POUs/FB_System.TcPOU
FUNCTION_BLOCK FB_System
VAR
	plcStart : PLC_Start;
	plcStop : PLC_Stop;
	plcReset : PLC_Reset;
	
	tcRestart : TC_Restart;
	tcConfig : TC_Config;
END_VAR

{attribute 'TcRpcEnable'}
METHOD configTC : BOOL
VAR_INPUT
END_VAR
tcConfig(
	NETID:= , 
	SET:= TRUE, 
	TMOUT:= , 
	BUSY=> , 
	ERR=> , 
	ERRID=> );
	
tcConfig(
	NETID:= , 
	SET:= FALSE, 
	TMOUT:= , 
	BUSY=> , 
	ERR=> , 
	ERRID=> );
END_METHOD

{attribute 'TcRpcEnable'}
METHOD resetPLC : BOOL
VAR_INPUT
END_VAR
plcReset(
	NETID:= , 
	PORT:= 851, 
	RESET:= TRUE, 
	TMOUT:= , 
	BUSY=> , 
	ERR=> , 
	ERRID=> );
	
plcReset(
	NETID:= , 
	PORT:= 851, 
	RESET:= FALSE, 
	TMOUT:= , 
	BUSY=> , 
	ERR=> , 
	ERRID=> );
END_METHOD

{attribute 'TcRpcEnable'}
METHOD restartTC : BOOL
tcRestart(
	NETID:= , 
	RESTART:= TRUE, 
	TMOUT:= , 
	BUSY=> , 
	ERR=> , 
	ERRID=> );
	
tcRestart(
	NETID:= , 
	RESTART:= FALSE, 
	TMOUT:= , 
	BUSY=> , 
	ERR=> , 
	ERRID=> );
END_METHOD

{attribute 'TcRpcEnable'}
METHOD startPLC : BOOL
plcStart(
	NETID:= '', 
	PORT:= 851, 
	START:= TRUE, 
	TMOUT:= , 
	BUSY=> , 
	ERR=> , 
	ERRID=> );
	
plcStart(
	NETID:= '', 
	PORT:= 851, 
	START:= FALSE, 
	TMOUT:= , 
	BUSY=> , 
	ERR=> , 
	ERRID=> );
END_METHOD

{attribute 'TcRpcEnable'}
METHOD stopPLC : BOOL
plcStop(
	NETID:= '', 
	PORT:= 851, 
	STOP:= TRUE, 
	TMOUT:= , 
	BUSY=> , 
	ERR=> , 
	ERRID=> );
	
plcStop(
	NETID:= '', 
	PORT:= 851, 
	STOP:= FALSE, 
	TMOUT:= , 
	BUSY=> , 
	ERR=> , 
	ERRID=> );
END_METHOD

END_FUNCTION_BLOCK

// ---- POUs/MAIN.TcPOU
PROGRAM MAIN
VAR
	moduleWB : WoodBunkEx;
	moduleCIP : ChipboardEx;
END_VAR

CallHardware(); //start program with hardware call - pass values and arrays into function blocks
SetupHardware(); //initialize values

runModules(); //LLD

CallHardware(); //end program with hardware call

ACTION runModules:
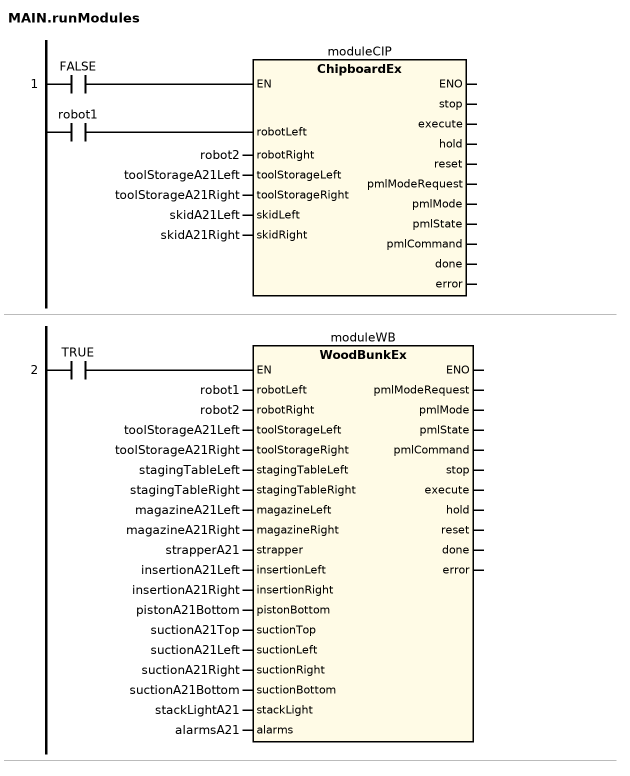
// NETWORK 1
IF FALSE THEN
    moduleCIP(
        robotLeft := robot1,
        robotRight := robot2,
        toolStorageLeft := toolStorageA21Left,
        toolStorageRight := toolStorageA21Right,
        skidLeft := skidA21Left,
        skidRight := skidA21Right); // ChipboardEx
END_IF

// NETWORK 2
moduleWB(
    robotLeft := robot1,
    robotRight := robot2,
    toolStorageLeft := toolStorageA21Left,
    toolStorageRight := toolStorageA21Right,
    stagingTableLeft := stagingTableLeft,
    stagingTableRight := stagingTableRight,
    magazineLeft := magazineA21Left,
    magazineRight := magazineA21Right,
    strapper := strapperA21,
    insertionLeft := insertionA21Left,
    insertionRight := insertionA21Right,
    pistonBottom := pistonA21Bottom,
    suctionTop := suctionA21Top,
    suctionLeft := suctionA21Left,
    suctionRight := suctionA21Right,
    suctionBottom := suctionA21Bottom,
    stackLight := stackLightA21,
    alarms := alarmsA21); // WoodBunkEx
END_ACTION

END_PROGRAM

// ---- POUs/A21b - Wood Bunk/WoodBunkEx.TcPOU
FUNCTION_BLOCK WoodBunkEx
VAR_IN_OUT //references to required hardware
	robotLeft, robotRight : RobotA21;
	toolStorageLeft, toolStorageRight : A21ToolStorage;
	
	stagingTableLeft, stagingTableRight : StagingTable;
	magazineLeft, magazineRight : SkidMagazine;
	
	strapper : StrapMachine;
	
	insertionLeft, insertionRight : Insertion;
	pistonBottom : SimplePiston;
	
	suctionTop : ARRAY[*] OF SuctionPad; (*1..3*)
	suctionLeft : ARRAY[*] OF SuctionPad; (*1..4*)
	suctionRight : ARRAY[*] OF SuctionPad; (*1..4*)
	suctionBottom : ARRAY[*] OF SuctionPad; (*1..2*)
	
	stackLight : PMLStackLight;
	alarms : A21Alarms;
END_VAR
VAR_OUTPUT //controls
	pmlModeRequest : E_PMLProtectedUnitMode := ePMLProtUnitMode_Maintenance;
	pmlMode : E_PMLProtectedUnitMode;
	
	pmlState : E_PMLState;
	pmlCommand : E_PMLCommand;

	stop : BOOL;
	execute : BOOL;
	hold : BOOL;
	reset : BOOL;
	
	done : BOOL;
	error : BOOL;
END_VAR
VAR
	pmlModeString : STRING;
	pmlStateString : STRING;
	
	pmlStateMachine : PML_StateMachine;
	pmlModeManager : PML_UnitModeManager;

	step : (IDLE, STAGING, LOAD_WB, PUSH, STRAP, RELEASE, COMPLETE := 1050);
	iPair : INT;
	
	stageStepLeft, stageStepRight : INT;
	loadStepLeft, loadStepRight : INT;
END_VAR
VAR //local types	
	demoHeight : REAL := 640; //mm
	materialsArr : ARRAY[0..GVL.maxPairs] OF PositionMaterials := [
		( position := 0, top := 'WDS20', left := 'WDS20', right := 'WDS20', bottom := 'WDB20' )];
		//( position := 69, top := 'WDS20', left := 'WDS20', right := 'WDS20', bottom := 'WDB20' )];
	
	loadedMaterials : ARRAY[Surface.TOP..Surface.BOTTOM] OF STRING;
END_VAR
VAR CONSTANT
	sectionID : SectionEnum := SectionEnum.WOOD_BUNK;
	suctionReleaseDelay : TIME := T#1000MS;
END_VAR
VAR
	//AOIs encapsulate functionality and reduce the number of module variables
	aoiTemplateLeft, aoiTemplateRight : AOI_StagingTemplate;
	aoiStageLeft, aoiStageRight : AOI_StageWoodBunk; 
	aoiLoadLeft, aoiLoadRight : AOI_LoadWoodBunk;
	
	suctionRelease : TON;
	
	//for testing, to be removed when deployoed
	latchLeft, latchRight : BOOL; //prevents SMC sliders from overshooting
	suctionEnableTop, suctionEnableLeft, suctionEnableRight, suctionEnableBottom : BOOL;
END_VAR

initModules(); //initialize modules

blocks(); //call AOIs and large library FBs

runPML(); //run PackML state machine

ACTION blocks:
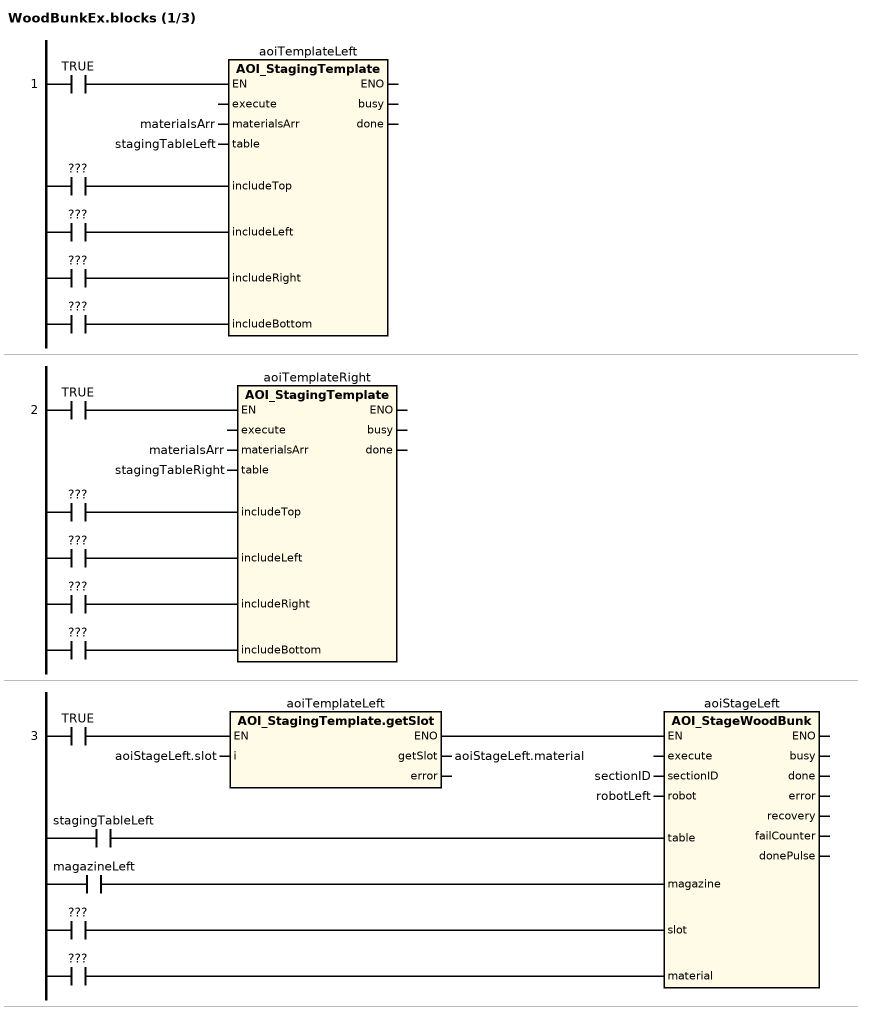
// NETWORK 1
aoiTemplateLeft(materialsArr := materialsArr, table := stagingTableLeft); // AOI_StagingTemplate

// NETWORK 2
aoiTemplateRight(materialsArr := materialsArr, table := stagingTableRight); // AOI_StagingTemplate

// NETWORK 3
aoiTemplateLeft.getSlot(i := aoiStageLeft.slot, getSlot => aoiStageLeft.material);
aoiStageLeft(sectionID := sectionID, robot := robotLeft, table := stagingTableLeft, magazine := magazineLeft); // AOI_StageWoodBunk

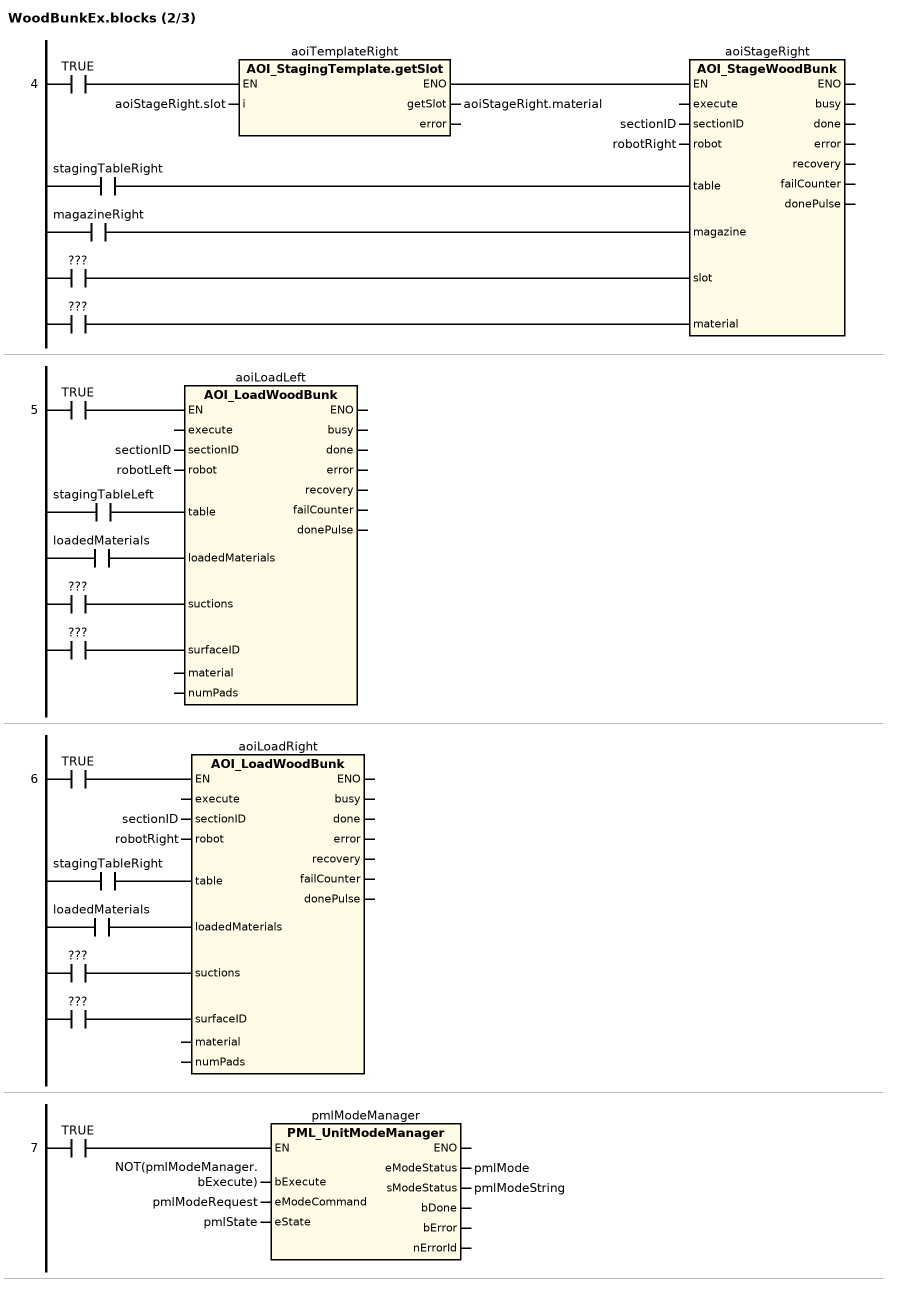
// NETWORK 4
aoiTemplateRight.getSlot(i := aoiStageRight.slot, getSlot => aoiStageRight.material);
aoiStageRight(
    sectionID := sectionID,
    robot := robotRight,
    table := stagingTableRight,
    magazine := magazineRight); // AOI_StageWoodBunk

// NETWORK 5
aoiLoadLeft(
    sectionID := sectionID,
    robot := robotLeft,
    table := stagingTableLeft,
    loadedMaterials := loadedMaterials); // AOI_LoadWoodBunk

// NETWORK 6
aoiLoadRight(
    sectionID := sectionID,
    robot := robotRight,
    table := stagingTableRight,
    loadedMaterials := loadedMaterials); // AOI_LoadWoodBunk

// NETWORK 7
pmlModeManager(
    bExecute := NOT(pmlModeManager.bExecute),
    eModeCommand := pmlModeRequest,
    eState := pmlState,
    eModeStatus => pmlMode,
    sModeStatus => pmlModeString); // PML_UnitModeManager

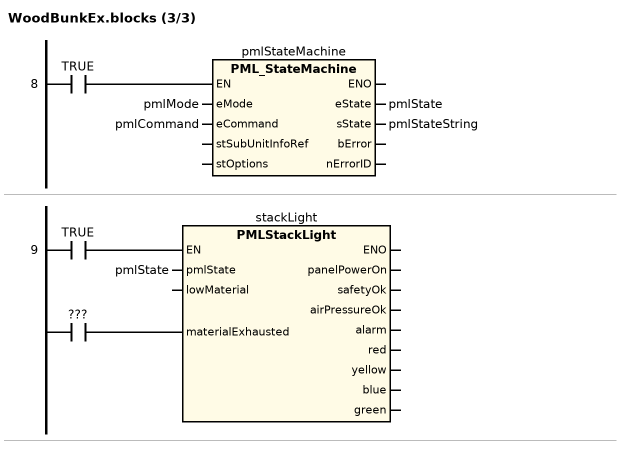
// NETWORK 8
pmlStateMachine(eMode := pmlMode, eCommand := pmlCommand, eState => pmlState, sState => pmlStateString); // PML_StateMachine

// NETWORK 9
stackLight(pmlState := pmlState); // PMLStackLight
END_ACTION

ACTION initModules:
{warning disable C0371}

stackLight.pmlState := pmlState;
//stackLight.lowMaterial := FALSE;
//stackLight.materialExhausted := FALSE;
END_ACTION

METHOD PRIVATE load : BOOL
VAR_INPUT
	pairIndex : INT;
END_VAR
VAR_OUTPUT
	error : BOOL;
END_VAR
VAR
	pair : REFERENCE TO PositionMaterials REF= materialsArr[pairIndex];
	errorLeft, errorRight : BOOL;
END_VAR
{warning disable C0371}
(*
this is the new code for loading wood bunks from staging table to insertion
loading sequences are independent as each side has its own step variable
can be extended by changing the include<> parameters
*)

load :=
	loadEx(
		robot:= robotLeft, 
		aoiLoad:= aoiLoadLeft, 
		loadStep:= loadStepLeft, 
		pairIndex:= pairIndex, 
		includeTop:= TRUE, 
		includeLeft:= TRUE, 
		includeRight:= FALSE, 
		includeBottom:= FALSE, 
		error=> errorLeft)
	AND
	loadEx(
		robot:= robotRight, 
		aoiLoad:= aoiLoadRight, 
		loadStep:= loadStepRight, 
		pairIndex:= pairIndex, 
		includeTop:= FALSE, 
		includeLeft:= FALSE, 
		includeRight:= TRUE, 
		includeBottom:= TRUE, 
		error=> errorRight);
		
error := errorLeft OR errorRight;

(*
below is the old code for loading wood bunks from staging table to insertion
it loads wood bunks in sets - top/bottom, then sides
if one side is finished loading a set before the other, it waits until the other side is done before advancing the set
*)
(*
IF robotLeft.error OR robotRight.error THEN
	error := TRUE;
	RETURN;
	
ELSIF 
	(robotLeft.reservation <> sectionID AND_THEN NOT robotLeft.reserve(sectionID)) OR 
	(robotRight.reservation <> sectionID AND_THEN NOT robotRight.reserve(sectionID))
THEN //loading requires both robots be reserved together
	RETURN;
	
ELSIF //robots have wrong tool
	(robotLeft.tool <> sectionID AND_THEN NOT robotLeft.changeEOAT(targetTool := sectionID)) OR
	(robotRight.tool <> sectionID AND_THEN NOT robotRight.changeEOAT(targetTool := sectionID))
THEN
	RETURN;
	
END_IF

CASE loadStep OF
	0: //top and bottom
		IF aoiLoadLeft.done AND aoiLoadRight.done THEN
			aoiLoadLeft.execute := aoiLoadRight.execute := FALSE;
			aoiLoadLeft.material := aoiLoadRight.material := '';
			
			aoiLoadLeft.reset();
			aoiLoadRight.reset();
			loadStep := 10;
			RETURN;
		END_IF
		
		aoiLoadLeft.suctions := suctionTop;
		aoiLoadLeft.surfaceID := Surface.TOP;
		aoiLoadLeft.material := pair.top;
		aoiLoadLeft.numPads := UPPER_BOUND(suctionTop, 1) - LOWER_BOUND(suctionTop, 1) + 1;
		
		aoiLoadRight.suctions := suctionBottom;
		aoiLoadRight.surfaceID := Surface.BOTTOM;
		aoiLoadRight.material := pair.bottom;
		aoiLoadRight.numPads := UPPER_BOUND(suctionBottom, 1) - LOWER_BOUND(suctionBottom, 1) + 1;
		
		aoiLoadLeft.execute := NOT aoiLoadLeft.done AND NOT aoiLoadLeft.busy;
		aoiLoadRight.execute := NOT aoiLoadRight.done AND NOT aoiLoadRight.busy;
		
	10: //sides
		IF aoiLoadLeft.done AND aoiLoadRight.done THEN
			aoiLoadLeft.execute := aoiLoadRight.execute := FALSE;
			aoiLoadLeft.material := aoiLoadRight.material := '';
			
			aoiLoadLeft.reset();
			aoiLoadRight.reset();
			loadStep := COMPLETE;
			RETURN;
		END_IF
		
		aoiLoadLeft.suctions := suctionLeft;
		aoiLoadLeft.surfaceID := Surface.LEFT;
		aoiLoadLeft.material := pair.left;
		aoiLoadLeft.numPads := UPPER_BOUND(suctionLeft, 1) - LOWER_BOUND(suctionLeft, 1) + 1;
		
		aoiLoadRight.suctions := suctionRight;
		aoiLoadRight.surfaceID := Surface.RIGHT;
		aoiLoadRight.material := pair.right;
		aoiLoadRight.numPads := UPPER_BOUND(suctionRight, 1) - LOWER_BOUND(suctionRight, 1) + 1;
		
		aoiLoadLeft.execute := NOT aoiLoadLeft.done AND NOT aoiLoadLeft.busy;
		aoiLoadRight.execute := NOT aoiLoadRight.done AND NOT aoiLoadRight.busy;
		
	COMPLETE:				
		robotLeft.release(sectionID);
		robotRight.release(sectionID);
		
		aoiLoadLeft.material := aoiLoadRight.material := '';
		aoiLoadLeft.execute := aoiLoadRight.execute := FALSE;
		
		loadStep := 0;
		load := TRUE;
END_CASE

//--------------------------------------------------
IF aoiLoadLeft.recovery THEN //if loading in recovery mode - refill table, resume loading when finished
	aoiLoadLeft.execute := stageEx(
		robot:= robotLeft, 
		aoiTemplate:= aoiTemplateLeft, 
		aoiStaging:= aoiStageLeft, 
		stageStep:= stageStepLeft, 
		includeTop:= TRUE, 
		includeLeft:= TRUE, 
		includeRight:= FALSE, 
		includeBottom:= FALSE, 
		error=> );
ELSE
	//loadLeft.execute := NOT loadLeft.busy AND NOT loadLeft.done;
END_IF
//--------------------------------------------------
IF aoiLoadRight.recovery THEN
	aoiLoadRight.execute := stageEx(
		robot:= robotRight, 
		aoiTemplate:= aoiTemplateRight, 
		aoiStaging:= aoiStageRight, 
		stageStep:= stageStepRight, 
		includeTop:= FALSE, 
		includeLeft:= FALSE, 
		includeRight:= TRUE, 
		includeBottom:= TRUE, 
		error=> );
ELSE
	//loadRight.execute := NOT loadRight.busy AND NOT loadRight.done;
END_IF
//--------------------------------------------------
	
error := aoiLoadLeft.error OR aoiLoadRight.error;
*)
END_METHOD

METHOD PRIVATE loadEx : BOOL
VAR_IN_OUT
	robot : RobotA21;
	aoiLoad : AOI_LoadWoodBunk;
	loadStep : INT;
END_VAR
VAR_INPUT
	pairIndex : INT;
	includeTop, includeLeft, includeRight, includeBottom : BOOL;
END_VAR
VAR_OUTPUT
	error : BOOL;
END_VAR
VAR
	pair : REFERENCE TO PositionMaterials REF= materialsArr[pairIndex];
END_VAR
{warning disable C0371}
IF robot.error THEN
	error := TRUE;
	RETURN;
ELSIF robot.reservation <> sectionID AND_THEN NOT robot.reserve(sectionID) THEN
	RETURN;
ELSIF robot.tool <> sectionID AND_THEN NOT robot.changeEOAT(targetTool := sectionID) THEN
	RETURN;
END_IF

error := aoiLoad.error;

CASE loadStep OF
	0:
		loadStep := Surface.TOP;
	
	Surface.TOP:		
		IF NOT includeTop OR aoiLoad.donePulse THEN
			aoiLoad.execute := FALSE;
			aoiLoad.material := '';
			loadStep := Surface.BOTTOM;
			RETURN;
		END_IF
		
		aoiLoad.surfaceID := Surface.TOP;
		aoiLoad.material := pair.top;
		aoiLoad.suctions := suctionTop;
		aoiLoad.numPads := UPPER_BOUND(suctionTop, 1) - LOWER_BOUND(suctionTop, 1) + 1;
		
		aoiLoad.execute := NOT aoiLoad.busy;
		
	Surface.BOTTOM:
		IF NOT includeBottom OR aoiLoad.donePulse THEN
			aoiLoad.execute := FALSE;
			aoiLoad.material := '';
			loadStep := Surface.LEFT;
			RETURN;
		END_IF
		
		aoiLoad.surfaceID := Surface.BOTTOM;
		aoiLoad.material := pair.bottom;
		aoiLoad.suctions := suctionBottom;
		aoiLoad.numPads := UPPER_BOUND(suctionBottom, 1) - LOWER_BOUND(suctionBottom, 1) + 1;
		
		aoiLoad.execute := NOT aoiLoad.busy;
		
	Surface.LEFT:
		IF NOT includeLeft OR aoiLoad.donePulse THEN
			aoiLoad.execute := FALSE;
			aoiLoad.material := '';
			loadStep := Surface.RIGHT;
			RETURN;
		END_IF
		
		aoiLoad.surfaceID := Surface.LEFT;
		aoiLoad.material := pair.left;
		aoiLoad.suctions := suctionLeft;
		aoiLoad.numPads := UPPER_BOUND(suctionLeft, 1) - LOWER_BOUND(suctionLeft, 1) + 1;
		
		aoiLoad.execute := NOT aoiLoad.busy;
		
	Surface.RIGHT:
		IF NOT includeRight OR aoiLoad.donePulse THEN
			aoiLoad.execute := FALSE;
			aoiLoad.material := '';
			loadStep := COMPLETE;
			RETURN;
		END_IF
		
		aoiLoad.surfaceID := Surface.RIGHT;
		aoiLoad.material := pair.right;
		aoiLoad.suctions := suctionRight;
		aoiLoad.numPads := UPPER_BOUND(suctionRight, 1) - LOWER_BOUND(suctionRight, 1) + 1;
		
		aoiLoad.execute := NOT aoiLoad.busy;
		
	COMPLETE:				
		robot.release(sectionID);
		
		aoiLoad.material := '';
		aoiLoad.execute := FALSE;
		
		loadEx := TRUE;
END_CASE
END_METHOD

METHOD PRIVATE maintenance : BOOL
VAR_INPUT
END_VAR
{warning disable C0371}
//no specific tasks yet, free run and testing
SetSuctions(suctionTop, suctionEnableTop);
SetSuctions(suctionLeft, suctionEnableLeft);
SetSuctions(suctionRight, suctionEnableRight);
SetSuctions(suctionBottom, suctionEnableBottom);

IF robotLeft.Done THEN
	robotLeft.clearCommand();
END_IF

IF robotRight.Done THEN
	robotRight.clearCommand();
END_IF
END_METHOD

METHOD PRIVATE process : BOOL
VAR_INPUT
	manualMode : BOOL;
END_VAR
VAR_OUTPUT
	error : BOOL;
END_VAR
{warning disable C0371}
suctionRelease(IN:= , PT:= suctionReleaseDelay, Q=> , ET=> );

CASE step OF
	IDLE:
		step := STAGING;
		
	STAGING:
		IF NOT done THEN
			done := stage(); //calls stageEx() for both robots
		END_IF
		
		IF
			(manualMode AND_THEN execute) OR
			(NOT manualMode AND_THEN done)
		THEN
			robotLeft.clearCommand();
			robotRight.clearCommand();
			
			aoiStageLeft.reset();
			aoiStageRight.reset();
			
			stageStepLeft := stageStepRight := 0;
			
			execute := FALSE;
			done := FALSE;
			step := LOAD_WB;
		END_IF
	
	LOAD_WB:
		IF NOT done THEN
			done := load(pairIndex := iPair, error => error);
		END_IF
		
		IF manualMode THEN
			SetSuctions(suctionTop, suctionEnableTop);
			SetSuctions(suctionLeft, suctionEnableLeft);
			SetSuctions(suctionRight, suctionEnableRight);
			SetSuctions(suctionBottom, suctionEnableBottom);
		END_IF
		
		IF
			(manualMode AND_THEN execute) OR
			(NOT manualMode AND_THEN done)
		THEN
			robotLeft.clearCommand();
			robotRight.clearCommand();
			
			aoiLoadLeft.reset();
			aoiLoadRight.reset();
			
			loadStepLeft := loadStepRight := 0;
			stageStepLeft := stageStepRight := 0;
			
			done := FALSE;
			suctionEnableTop := suctionEnableLeft := suctionEnableRight := suctionEnableBottom := FALSE;
			execute := FALSE;
			
			step := PUSH;
		END_IF
		
	PUSH:
		IF
			(manualMode AND_THEN execute) OR
			(NOT manualMode AND latchLeft AND latchRight AND pistonBottom.extended)
		THEN
			insertionLeft.stop();
			insertionRight.stop();
			
			latchLeft := latchRight := FALSE;
			execute := FALSE;
			step := STRAP;
			RETURN;
		END_IF
		
		IF NOT validateInsertion(checkTop:= FALSE, checkLeft:= FALSE, checkRight:= FALSE, checkBottom:= FALSE) THEN
			error := TRUE;
			RETURN;
		END_IF
		
		insertionLeft.align(targetPos := demoHeight/2);
		insertionRight.align(targetPos := demoHeight/2);
		
		IF
			insertionLeft.sliderPos <> demoHeight/2 OR 
			insertionRight.sliderPos <> demoHeight/2
		THEN
			RETURN;
		END_IF
		
		IF NOT latchLeft THEN
			latchLeft := insertionLeft.contact;
			insertionLeft.press();
		END_IF
		
		IF NOT latchRight THEN
			latchRight := insertionRight.contact;
			insertionRight.press();
		END_IF
		
		(*
		IF insertionLeft.contact THEN
			latchLeft := TRUE;
		ELSIF NOT latchLeft THEN
			insertionLeft.press();
		END_IF
		
		IF insertionRight.contact THEN
			latchRight := TRUE;
		ELSIF NOT latchRight THEN
			insertionRight.press();
		END_IF
		*)
		pistonBottom.extend();
		
	STRAP:	
		strapper.bEnable := TRUE;
		IF strapper.done THEN
			suctionRelease.IN := FALSE;
			step := RELEASE;
			RETURN;
		END_IF
		
		IF suctionRelease.Q THEN
			SetSuctions(suctionTop, FALSE);
			SetSuctions(suctionLeft, FALSE);
			SetSuctions(suctionRight, FALSE);
			SetSuctions(suctionBottom, FALSE);
		ELSIF strapper.atBundleLevel THEN
			suctionRelease.IN := TRUE;
		END_IF
		
		IF strapper.ready THEN
			strapper.strap();
		END_IF
		
		IF execute THEN
			suctionRelease.IN := FALSE;
			execute := FALSE;
			step := RELEASE;
		END_IF
		
	RELEASE: //release command		
		//insertionLeft.align(0);
		//insertionRight.align(0);
		//insertionLeft.release();
		//insertionRight.release();
		insertionLeft.toHome();
		insertionRight.toHome();
		
		pistonBottom.retract();
		
		IF 
			(insertionLeft.screw.AtHome AND insertionRight.screw.AtHome AND pistonBottom.retracted) OR
			execute
		THEN
			execute := FALSE;
			step := COMPLETE;
		END_IF
	
	COMPLETE:
		//reset everything
		iPair := (iPair + 1) MOD GVL.maxPairs;
		step := IDLE;
		
		process := TRUE;
END_CASE
END_METHOD

METHOD PRIVATE ps_Aborting : BOOL
VAR_INPUT
END_VAR
{warning disable C0371}
insertionLeft.stop();
insertionRight.stop();
pistonBottom.stop();

aoiLoadLeft.reset();
aoiLoadRight.reset();

aoiStageLeft.reset();
aoiStageRight.reset();

robotLeft.clearCommand();
robotRight.clearCommand();

//stop conveyors

ps_Aborting :=
	NOT insertionLeft.active AND
	NOT insertionRight.active AND
	NOT pistonBottom.busy AND
	NOT robotLeft.Busy AND
	NOT robotRight.Busy;
END_METHOD

METHOD PRIVATE ps_Clearing : BOOL
VAR_INPUT
END_VAR
{warning disable C0371}
insertionLeft.reset();
insertionRight.reset();

ps_Clearing := 
	NOT insertionLeft.error AND
	NOT insertionRight.error AND
	NOT strapper.error AND
	NOT robotLeft.error AND
	NOT robotRight.error AND
	NOT strapper.error;
END_METHOD

METHOD PRIVATE ps_Execute : BOOL
VAR_INPUT
END_VAR
VAR_OUTPUT
	error : BOOL;
END_VAR
CASE pmlMode OF
	0: //invalid mode
	ePMLProtUnitMode_Production:	ps_Execute := process(manualMode := FALSE, error => error);
	ePMLProtUnitMode_Maintenance:	maintenance();
	ePMLProtUnitMode_Manual:		ps_Execute := process(manualMode := TRUE, error => error);
END_CASE
END_METHOD

METHOD PRIVATE ps_Holding : BOOL
VAR_INPUT
END_VAR
{warning disable C0371}
insertionLeft.stop();
insertionRight.stop();
pistonBottom.stop();
//set robot to pause

ps_Holding :=
	NOT insertionLeft.active AND
	NOT insertionRight.active;
END_METHOD

METHOD PRIVATE ps_Resetting : BOOL
VAR_INPUT
END_VAR
{warning disable C0371}
insertionLeft.reset();
insertionRight.reset();

ps_Resetting := 
	reset AND
	NOT insertionLeft.error AND
	NOT insertionRight.error AND
	NOT strapper.error AND
	NOT robotLeft.error AND
	NOT robotRight.error;
END_METHOD

METHOD PRIVATE ps_Starting : BOOL
VAR_INPUT
END_VAR
{warning disable C0371}
robotLeft.clearCommand();
robotRight.clearCommand();

insertionLeft.homingSequence();
insertionRight.homingSequence();
pistonBottom.retract();

ps_Starting := 
	insertionLeft.homingComplete AND 
	insertionRight.homingComplete AND 
	pistonBottom.retracted;
END_METHOD

METHOD PRIVATE ps_Stopping : BOOL
VAR_INPUT
END_VAR
{warning disable C0371}
insertionLeft.stop();
insertionRight.stop();
pistonBottom.stop();

aoiLoadLeft.reset();
aoiLoadRight.reset();

aoiStageLeft.reset();
aoiStageRight.reset();

robotLeft.clearCommand();
robotRight.clearCommand();

//stop conveyors

ps_Stopping :=
	NOT insertionLeft.active AND
	NOT insertionRight.active AND
	NOT pistonBottom.busy AND
	NOT robotLeft.Busy AND
	NOT robotRight.Busy;
END_METHOD

ACTION runPML:
(*
PackML
	state machine for packaging applications - see Tc3_PackML_V2 library on InfoSys
	
	final states - wait for an input or condition and command to new state
	intermediate states - complete a task and call pmlStateMachine.M_StateComplete() to advance to next state
	
the following states currently use the same logic (albeit in different methods), implementation may change later
	ps_Stopping() and ps_Aborting()
	ps_Resetting() and ps_Clearing()
	
STOP - controlled stop induced by operator/HMI **with intent to shut down or change mode** - otherwise use HOLD
ABORT - emergency stop due to machine errors


HOLD - minor local issues
SUSPEND - external issues

EXECUTE - major control logic
	different modes may require different tasks
	create methods as required for different modes, then call the correct method in ps_Completing()
	can be commanded to STOP, ABORT, HOLD, or SUSPEND at any point
COMPLETING - process complete, move product out of system and finish transition to COMPLETED
*)

(*
IF //abort at machine error
	insertionLeft.error OR 
	insertionRight.error OR 
	robotLeft.error OR 
	robotRight.error OR
	strapper.error
THEN
	pmlCommand := ePMLCommand_Abort;
	
ELSIF stop THEN //stop at command stop
	pmlCommand := ePMLCommand_Stop;

ELSIF FALSE (*A2.4 cannot allow bundles to enter*) THEN //FALSE condition never executes - this is temporary
	pmlCommand := ePMLCommand_Suspend;
END_IF
*)
IF stop THEN //stop at command stop
	pmlCommand := ePMLCommand_Stop;
END_IF

CASE pmlState OF
	0: (*ePMLState_Undefined*) //default state on startup
		pmlCommand := ePMLCommand_Stop;
		
	ePMLState_Stopping:
		IF ps_Stopping() THEN
			pmlStateMachine.M_StateComplete();
		END_IF
		
	ePMLState_Stopped:
		pmlCommand := ePMLCommand_Reset;
	
    ePMLState_Resetting:
		//IF ps_Resetting() THEN
			reset := FALSE;
			pmlStateMachine.M_StateComplete();
		//END_IF
		
	ePMLState_Idle:
		IF execute THEN
			execute := FALSE;
			pmlCommand := ePMLCommand_Start;
		END_IF		
	
	ePMLState_Starting:
		IF ps_Starting() THEN
			pmlStateMachine.M_StateComplete();
		END_IF
	
	ePMLState_Execute: 
		IF hold THEN
			pmlCommand := ePMLCommand_Hold;
		END_IF
		
		IF ps_Execute(error => error) THEN
			pmlStateMachine.M_StateComplete();
			pmlCommand := ePMLCommand_Complete;
		END_IF
		
	ePMLState_Completing:
		pmlStateMachine.M_StateComplete();
	
	ePMLState_Complete:
		pmlCommand := ePMLCommand_Reset;
	
	ePMLState_Holding:
		IF ps_Holding() THEN
			pmlStateMachine.M_StateComplete();
		END_IF
	
	ePMLState_Held:
		IF NOT hold THEN
			pmlCommand := ePMLCommand_Unhold;
		END_IF
	
	ePMLState_Unholding:
		pmlStateMachine.M_StateComplete(); //release all pause commands and IO
	
	ePMLState_Suspended: //based on output section conditions
	ePMLState_Suspending: //based on output section conditions
	ePMLState_Unsuspending: //based on output section conditions
	
	ePMLState_Aborting:
		IF ps_Aborting() THEN
			pmlStateMachine.M_StateComplete();
		END_IF
	
	ePMLState_Aborted:
		pmlCommand := ePMLCommand_Clear;
	
	ePMLState_Clearing:
		IF ps_Clearing() THEN
			pmlStateMachine.M_StateComplete();
		END_IF
	
END_CASE
END_ACTION

METHOD PRIVATE stage : BOOL
VAR_OUTPUT
	error : BOOL;
END_VAR
{warning disable C0371}

(*
this method only exists to call stageEx() for both robots
*)
(*
stage := leftDone AND rightDone;

IF NOT leftDone THEN
	leftDone := stageEx(
		robot:= robotLeft, 
		aoiTemplate:= aoiTemplateLeft, 
		aoiStaging:= aoiStageLeft, 
		stageStep:= stageStepLeft, 
		//iSlot:= iSlotLeft, 
		includeTop:= TRUE, 
		includeLeft:= TRUE, 
		includeRight:= FALSE, 
		includeBottom:= FALSE, 
		error=> );
END_IF

IF NOT rightDone THEN
	rightDone := stageEx(
		robot:= robotRight, 
		aoiTemplate:= aoiTemplateRight, 
		aoiStaging:= aoiStageRight, 
		stageStep:= stageStepRight, 
		//iSlot:= iSlotRight, 
		includeTop:= FALSE, 
		includeLeft:= FALSE, 
		includeRight:= TRUE, 
		includeBottom:= TRUE, 
		error=> );
END_IF
*)

stage := 
	stageEx(
		robot:= robotLeft, 
		aoiTemplate:= aoiTemplateLeft, 
		aoiStaging:= aoiStageLeft, 
		stageStep:= stageStepLeft, 
		includeTop:= TRUE, 
		includeLeft:= TRUE, 
		includeRight:= FALSE, 
		includeBottom:= FALSE, 
		error=> )
	AND
	stageEx(
		robot:= robotRight, 
		aoiTemplate:= aoiTemplateRight, 
		aoiStaging:= aoiStageRight, 
		stageStep:= stageStepRight, 
		includeTop:= FALSE, 
		includeLeft:= FALSE, 
		includeRight:= TRUE, 
		includeBottom:= TRUE, 
		error=> );
END_METHOD

METHOD PRIVATE stageEx : BOOL
VAR_IN_OUT
	robot : RobotA21;
	aoiTemplate : AOI_StagingTemplate;
	aoiStaging : AOI_StageWoodBunk;
	stageStep : INT;
END_VAR
VAR_INPUT
	includeTop, includeLeft, includeRight, includeBottom : BOOL;
END_VAR
VAR_OUTPUT
	error : BOOL;
END_VAR
{warning disable C0371}
IF robot.error THEN
	error := TRUE;
	RETURN;
ELSIF robot.reservation <> sectionID AND_THEN NOT robot.reserve(sectionID) THEN
	RETURN;
ELSIF robot.tool <> sectionID AND_THEN NOT robot.changeEOAT(targetTool := sectionID) THEN
	RETURN;
END_IF

CASE stageStep OF
	0: //generate staging template
		IF aoiTemplate.done THEN
			aoiTemplate.execute := FALSE;
			stageStep := 10;
			RETURN;
		END_IF
		
		aoiTemplate.execute := NOT aoiTemplate.busy;
		
		aoiTemplate.includeTop := includeTop;
		aoiTemplate.includeLeft := includeLeft;
		aoiTemplate.includeRight := includeRight;
		aoiTemplate.includeBottom := includeBottom;
		
	10: //stage tables
		IF aoiStaging.slot > 10 THEN
			aoiStaging.execute := FALSE;			
			stageStep := COMPLETE;
			RETURN;
		END_IF
		
		aoiStaging.execute := NOT aoiStaging.busy; //execute if aoiStaging is ready
		
		aoiStaging.slot := MAX(1, aoiStaging.slot); //if 0, sets to 1
		aoiStaging.slot := MIN(aoiStaging.slot, 999); //prevents overflow 
		
		IF aoiStaging.donePulse THEN
			aoiStaging.slot := aoiStaging.slot + 1;
		END_IF
	
	COMPLETE:
		aoiTemplate.clearTemplate();
		aoiTemplate.execute := FALSE;
		aoiStaging.execute := FALSE;
		aoiStaging.reset();
		
		robot.release(sectionID);
		
		aoiStaging.slot := 0;
		
		stageEx := TRUE;
		//stageStep := 0;
END_CASE

error := aoiStaging.error;
END_METHOD

METHOD PRIVATE validateInsertion : BOOL
VAR_INPUT
	checkTop : BOOL;
	checkLeft : BOOL;
	checkRight : BOOL;
	checkBottom : BOOL;
END_VAR
validateInsertion := 
	(NOT checkTop OR_ELSE SuctionQuality(suctions:= suctionTop)) AND
	(NOT checkLeft OR_ELSE SuctionQuality(suctions:= suctionLeft)) AND
	(NOT checkRight OR_ELSE SuctionQuality(suctions:= suctionRight)) AND
	(NOT checkBottom OR_ELSE SuctionQuality(suctions:= suctionBottom));

(*
validateSuctionQuality := 
	(
		NOT checkTop OR_ELSE InsertionQuality(
			suctions:= suctionTop, 
			insertionMaterial:= loadedMaterials[Surface.TOP], 
			recipeMaterial:= materialsArr[iPair].top)
	) AND
	(
		NOT checkLeft OR_ELSE InsertionQuality(
			suctions:= suctionLeft, 
			insertionMaterial:= loadedMaterials[Surface.LEFT], 
			recipeMaterial:= materialsArr[iPair].left)
	) AND
	(
		NOT checkRight OR_ELSE InsertionQuality(
			suctions:= suctionRight, 
			insertionMaterial:= loadedMaterials[Surface.RIGHT], 
			recipeMaterial:= materialsArr[iPair].right)
	) AND
	(
		NOT checkBottom OR_ELSE InsertionQuality(
			suctions:= suctionBottom, 
			insertionMaterial:= loadedMaterials[Surface.BOTTOM], 
			recipeMaterial:= materialsArr[iPair].bottom)
	);
*)
END_METHOD

END_FUNCTION_BLOCK

// ---- POUs/A21b - Wood Bunk/AOIs/AOI_StagingTemplate.TcPOU
FUNCTION_BLOCK AOI_StagingTemplate
VAR_INPUT
	execute : BOOL;
END_VAR
VAR_IN_OUT
	materialsArr : ARRAY[*] OF PositionMaterials; //[0..GVL.maxPairs]
	table : StagingTable;
END_VAR
VAR_INPUT
	includeTop, includeLeft, includeRight, includeBottom : BOOL; 
END_VAR
VAR_OUTPUT
	busy : BOOL;
	done : BOOL;
END_VAR
VAR
	trigger : R_TRIG;
	run : BOOL;
	step : (IDLE, GENERATE_ARRAY, GENERATE_TEMPLATE, COMPLETE);
	i : INT;
END_VAR
VAR	
	stagingArray : ARRAY[0..(GVL.maxPairs+1)*2] OF STRING;
	
	template : StagingTable;
	templateSlots AT %M* : ARRAY[1..10] OF MaterialSlot;
END_VAR

{warning disable C0371}
(*
this AOI can be implemented without steps, but doing so should shorten PLC cycles
*)

template(slots:= templateSlots);

trigger(CLK:= execute, Q=> run);
busy := run OR step > 0;

CASE step OF
	IDLE:
		IF run THEN
			step := GENERATE_ARRAY;
			done := FALSE;
		END_IF
		
	GENERATE_ARRAY:
		//strings contain garbage chars after a null byte, they must be manually cleaned before checking if they are byte-empty
		CleanStringsArray(arr := stagingArray);
		IF ArrayIsEmpty(arr := ADR(stagingArray), arrSize := SIZEOF(stagingArray)) THEN //if staging array is empty, fill the array
			createStagingArray(
				includeTop:= includeTop, 
				includeLeft:= includeLeft, 
				includeRight:= includeRight, 
				includeBottom:= includeBottom);
		END_IF
		
		step := GENERATE_TEMPLATE;
		
	GENERATE_TEMPLATE:
		//copy over the real slots before autofilling, otherwise the template may fill occupied slots
		table.copyFrom(src := table);
		
		(*
		iterate through all pairs and autofill the template
		replace succesfully autofilled materials with empty string
		if staging needs to be performed a 2nd time, autofilling empty strings is always unsuccessful
		*)
		FOR i:=0 TO (GVL.maxPairs+1)*2 BY 1 DO
			IF template.autofill(material := stagingArray[i]) THEN
				stagingArray[i] := '';
			END_IF
		END_FOR
		
		step := COMPLETE;
	
	COMPLETE:
		done := TRUE;
		
		step := IDLE;
		
END_CASE

METHOD PRIVATE addToStagingArray : BOOL
VAR_INPUT
	material : STRING;
END_VAR
VAR
	remainingMaterial : STRING;
	splitMaterial : STRING;
END_VAR
remainingMaterial := material;
WHILE FIND(remainingMaterial, '_') > 0 DO
	splitCombinedMaterials(remainingMaterial, splitMaterial);
	IF splitMaterial <> '' THEN
		AddToStringArray(arr := stagingArray, newString := splitMaterial, numElements => , nextIndex => );
		(*
		AddToArray(
			arr := ADR(stagingArray), 
			numEntries := SIZEOF(stagingArray)/SIZEOF(stagingArray[0]), 
			dataSize := SIZEOF(STRING), 
			newEntry := splitMaterial);
		*)
	END_IF
END_WHILE

IF remainingMaterial <> '' THEN
	AddToStringArray(arr := stagingArray, newString := remainingMaterial, numElements => , nextIndex => );
	(*
	AddToArray(
		arr := ADR(stagingArray), 
		numEntries := SIZEOF(stagingArray)/SIZEOF(stagingArray[0]), 
		dataSize := SIZEOF(STRING), 
		newEntry := remainingMaterial);
	*)
END_IF

addToStagingArray := TRUE;
END_METHOD

METHOD clearArray : BOOL
VAR_INPUT
END_VAR
MEMSET(ADR(stagingArray), 0, SIZEOF(stagingArray));
END_METHOD

METHOD clearTemplate : BOOL
VAR_INPUT
END_VAR
template.clear();
END_METHOD

METHOD PRIVATE createStagingArray : BOOL
VAR_INPUT
	includeTop : BOOL;
	includeLeft : BOOL;
	includeRight : BOOL;
	includeBottom : BOOL;
END_VAR
VAR
	remainingMaterial : STRING;
	splitMaterial : STRING;
	
	i : INT;
END_VAR
FOR i:=0 TO GVL.maxPairs BY 1 DO
	IF includeTop THEN
		addToStagingArray(material := materialsArr[i].top);
	END_IF
	
	IF includeLeft THEN
		addToStagingArray(material := materialsArr[i].left);
	END_IF
	
	IF includeRight THEN
		addToStagingArray(material := materialsArr[i].right);
	END_IF
	
	IF includeBottom THEN
		addToStagingArray(material := materialsArr[i].bottom);
	END_IF
END_FOR
END_METHOD

METHOD getSlot : STRING
VAR_INPUT
	i : INT;
END_VAR
VAR_OUTPUT
	error : BOOL;
END_VAR
getSlot := template.getSlot(i := i, error => error);
END_METHOD

METHOD reset : BOOL
VAR_INPUT
END_VAR
VAR
	temp : AOI_StagingTemplate;
END_VAR
//(*
busy := FALSE;
done := FALSE;
step := 0;

clearArray();
clearTemplate();
//*)
//THIS^ := temp;
END_METHOD

METHOD PRIVATE splitCombinedMaterials : BOOL
VAR_IN_OUT
	materialID : STRING;
	splitMaterial : STRING;
END_VAR
VAR
	i : INT;
END_VAR
FindAndSplitChar(
	sSeparatorChar:= '_', 
	pSrcString:= ADR(materialID), 
	
	pLeftString:= ADR(splitMaterial), 
	nLeftSize:= SIZEOF(splitMaterial), 
	
	pRightString:= ADR(materialID), 
	nRightSize:= SIZEOF(materialID), 
	
	bSearchFromRight:= FALSE);
END_METHOD

END_FUNCTION_BLOCK

// ---- POUs/Utility/ArrayIsEmpty.TcPOU
FUNCTION ArrayIsEmpty : BOOL
VAR_INPUT
	arr : POINTER TO BYTE;
	arrSize : LINT;
END_VAR
VAR
	i : LINT;
END_VAR

FOR i:=0 TO arrSize-1 BY 1 DO
	IF arr[i] <> 0 THEN
		RETURN;
	END_IF
END_FOR

ArrayIsEmpty := TRUE;

END_FUNCTION

// ---- POUs/A21a - Chipboard/ChipboardEx.TcPOU
FUNCTION_BLOCK ChipboardEx
VAR_IN_OUT //references to required hardware
	robotLeft, robotRight : RobotA21;
	toolStorageLeft, toolStorageRight : A21ToolStorage;
	
	skidLeft, skidRight : SkidMagazine;
END_VAR
VAR_OUTPUT //controls
	stop : BOOL;
	execute : BOOL;
	hold : BOOL;
	reset : BOOL;
	
	pmlModeRequest : E_PMLProtectedUnitMode := ePMLProtUnitMode_Production;
	pmlMode : E_PMLProtectedUnitMode;
	
	pmlState : E_PMLState;
	pmlCommand : E_PMLCommand;
END_VAR
VAR_OUTPUT
	done : BOOL;
	error : BOOL;
END_VAR
VAR
	pmlModeString : STRING;
	pmlStateString : STRING;
	
	pmlStateMachine : PML_StateMachine;
	pmlModeManager : PML_UnitModeManager;
	
	step : (IDLE, RETRACT_CONVEYOR, LOAD_CIP, EXTEND_CONVEYOR, COMPLETE := 1050);
	iPair : INT;
	
	loadSet : INT;
END_VAR
VAR //local types
	demoHeight : REAL := 600; //mm
	materialsArr : ARRAY[0..GVL.maxPairs] OF PositionMaterials := [
		(position := 0, top := 'CIP54', bottom := 'CIP18')
	];
		
	loadedMaterials : ARRAY[Surface.TOP..Surface.BOTTOM] OF STRING;
END_VAR
VAR CONSTANT
	sectionID : SectionEnum := SectionEnum.CHIPBOARD;
END_VAR
VAR
	aoiLoadLeft, aoiLoadRight : AOI_LoadChipboard;
	
	//for testing
	latchLeft, latchRight : BOOL;
END_VAR

{warning disable C0371}
callLocalModules(); //call local modules

blocks(); //call AOIs and large library FBs

runPML(); //run PackML state machine

ACTION blocks:
aoiLoadRight(
	sectionID:= sectionID, 
	execute:= ,
	robot:= robotRight, 
	storage:= skidRight,
	loadedMaterials:= loadedMaterials,
	surfaceID:= , 
	material:= , 
	loadedMaterials=> , 
	done=> , 
	error=> );
	
aoiLoadRight(
	sectionID:= sectionID, 
	execute:= , 
	robot:= robotRight, 
	storage:= skidRight,
	loadedMaterials:= loadedMaterials, 
	surfaceID:= , 
	material:= , 
	busy=> , 
	done=> , 
	error=> , 
	recovery=> , 
	failCounter=> );
END_ACTION

METHOD PRIVATE callLocalModules : BOOL
END_METHOD

METHOD PRIVATE load : BOOL
VAR_INPUT
	pairIndex : INT;
END_VAR
VAR_OUTPUT
	error : BOOL;
END_VAR
VAR
	pair : REFERENCE TO PositionMaterials REF= materialsArr[pairIndex];
END_VAR
{warning disable C0371}
IF robotLeft.error AND robotLeft.error THEN
	error := TRUE;
	RETURN;

ELSIF
	( robotLeft.reservation <> sectionID AND_THEN robotLeft.reserve(sectionID) ) OR
	( robotRight.reservation <> sectionID AND_THEN robotRight.reserve(sectionID) ) THEN
	RETURN;
	
ELSIF //wrong tool and not finished changing tool
	(robotLeft.tool <> sectionID AND_THEN NOT robotLeft.changeEOAT(targetTool := sectionID)) OR
	(robotRight.tool <> sectionID AND_THEN NOT robotRight.changeEOAT(targetTool := sectionID))
THEN
	RETURN;
END_IF
//robots ok

CASE loadSet OF
	0: //left robot -> top, right robot -> bottom
		IF aoiLoadLeft.done AND aoiLoadRight.done THEN
			aoiLoadLeft.execute := aoiLoadRight.execute := FALSE;
			loadSet := 10;
			RETURN;
		END_IF
		
		aoiLoadLeft.surfaceID := Surface.TOP;
		aoiLoadLeft.material := pair.left;
		
		aoiLoadRight.surfaceID := Surface.BOTTOM;
		aoiLoadRight.material := pair.right;
		
		aoiLoadLeft.execute := NOT aoiLoadLeft.recovery;
		aoiLoadRight.execute := NOT aoiLoadRight.recovery;
		
	10: //recovery		
		IF robotRight.error THEN //left ok, right error
			
			IF aoiLoadLeft.done THEN
				aoiLoadLeft.execute := FALSE;
				loadSet := COMPLETE;
				RETURN;
			END_IF
			
			aoiLoadLeft.surfaceID := Surface.BOTTOM;
			aoiLoadLeft.material := pair.bottom;
			aoiLoadLeft.execute := NOT aoiLoadLeft.recovery;
			
		ELSIF robotLeft.error THEN //left error, right ok
			
			IF aoiLoadRight.done THEN
				aoiLoadRight.execute := FALSE;
				loadSet := COMPLETE;
				RETURN;
			END_IF
			
			aoiLoadRight.surfaceID := Surface.TOP;
			aoiLoadRight.material := pair.top;
			aoiLoadRight.execute := NOT aoiLoadRight.recovery;
			
		END_IF
		
	COMPLETE:
		loadSet := 0;
		
		robotLeft.release(sectionID);
		robotRight.release(sectionID);
		
		load := TRUE;
END_CASE
END_METHOD

METHOD PRIVATE loadingSequence : BOOL
VAR_IN_OUT
	robot : RobotA21;
	storage : SkidMagazine;
	loadStep : INT;
END_VAR
VAR_INPUT
	surfaceID : Surface;
	material : STRING;
END_VAR
VAR_OUTPUT
	fail : BOOL;
END_VAR
VAR
	slot : INT;
END_VAR
VAR CONSTANT
	suctionDistance : INT := 10;
END_VAR
{warning disable C0371}
IF material = '' THEN
	loadingSequence := TRUE;
	RETURN;
END_IF

CASE loadStep OF
	0:
		robot.clearCommand();
		IF robot.Ready THEN
			loadStep := 1;
		END_IF
	
	1:
		IF surfaceID = Surface.BOTTOM (*AND_THEN conveyors not retracted*) THEN
			//retract conveyors
			RETURN;
		END_IF
		loadStep := 10;
		
	10: //grab from chipboard skid
		IF NOT storage.findSlot(material := material, index => slot) THEN
			fail := TRUE;
			RETURN;
		(*
		ELSIF surfaceID = Surface.BOTTOM (*AND_THEN (*conveyor not lowered*)*) THEN
			//lower conveyor
			RETURN;
		*)
		END_IF
		
		IF robot.eoatDistance < suctionDistance THEN
			robot.HoldMaterial := storage.getSlot(i := slot);
		END_IF
		
		IF robot.Done THEN
			loadStep := COMPLETE;
			RETURN;
		ELSIF robot.materialAtHoldingPosition.4 OR robot.materialAtHoldingPosition.5 THEN //bits 4 and 5 are chipboard in position
			loadStep := 20;
			RETURN;
		END_IF
		
		robot.setGroup(group := 1, value := A21.PLACE_CHIPBOARD_TOP);
		robot.setGroup(group := 2, value := slot);
		
	20: //place to bundle
		IF robotLeft.Done THEN
			loadStep := COMPLETE;
			RETURN;
		END_IF
		
		IF robot.HoldMaterial <> '' THEN
			loadedMaterials[surfaceID] := robot.HoldMaterial;
			robot.HoldMaterial := '';
		END_IF
		
	COMPLETE:
		IF loadedMaterials[surfaceID] = material THEN
			loadingSequence := TRUE;
		ELSE
			loadStep := 0;
		END_IF
		
END_CASE
END_METHOD

METHOD PRIVATE maintenance : BOOL
VAR_INPUT
END_VAR
{warning disable C0371}
//no specific tasks yet, free run and testing

IF robotLeft.Done THEN
	robotLeft.clearCommand();
END_IF

IF robotRight.Done THEN
	robotRight.clearCommand();
END_IF
END_METHOD

METHOD PRIVATE process : BOOL
VAR_INPUT
	manualMode : BOOL;
END_VAR
VAR_OUTPUT
	error : BOOL;
END_VAR
CASE step OF
	IDLE:
		IF execute THEN
			execute := FALSE;
			step := RETRACT_CONVEYOR;
		END_IF
		
	RETRACT_CONVEYOR:
		(*
		IF demoPair.bottom <> '' (*retract conveyors*) THEN
			IF TRUE (*BLSC 1-3 retracted*) THEN
				done := TRUE;
			END_IF
		ELSE
			done := TRUE;
		END_IF
		
		IF
			(manualStep AND_THEN execute) OR
			(NOT manualStep AND_THEN done)
		THEN
			done := FALSE;
			step := LOAD_MATERIAL;
		END_IF
		*)
		step := LOAD_CIP;
	LOAD_CIP:
		IF NOT done THEN
			done := load(pairIndex:= iPair, error=> error);
		END_IF
		
		IF
			(manualMode AND_THEN execute) OR
			(NOT manualMode AND_THEN done)
		THEN
			done := FALSE;
			execute := FALSE;
			
			step := EXTEND_CONVEYOR;
		END_IF
		
	EXTEND_CONVEYOR:
		(*
		IF FALSE (*conveyors not extended*) THEN
			//extend conveyors
		END_IF
		
		IF
			(manualStep AND_THEN execute) OR
			(FALSE) //conveyors extended
		THEN
			done := FALSE;
			step := COMPLETE;
		END_IF
		*)
		step := COMPLETE;
	COMPLETE:
		//reset everything
		step := IDLE;
		
		process := TRUE;
		
END_CASE
END_METHOD

METHOD PRIVATE ps_Aborting : BOOL
VAR_INPUT
END_VAR
{warning disable C0371}
aoiLoadLeft.reset();
aoiLoadRight.reset();

robotLeft.clearCommand();
robotRight.clearCommand();

//stop conveyors

ps_Aborting :=
	NOT robotLeft.Busy AND
	NOT robotRight.Busy;
END_METHOD

METHOD PRIVATE ps_Clearing : BOOL
VAR_INPUT
END_VAR
{warning disable C0371}
(*reset conveyors*)

ps_Clearing := 
	NOT robotLeft.error AND
	NOT robotRight.error;
END_METHOD

METHOD PRIVATE ps_Execute : BOOL
VAR_INPUT
END_VAR
VAR_OUTPUT
	error : BOOL;
END_VAR
CASE pmlMode OF
	0: //invalid mode
	ePMLProtUnitMode_Production:	ps_Execute := process(manualMode := FALSE, error => error);
	ePMLProtUnitMode_Maintenance:	maintenance();
	ePMLProtUnitMode_Manual:		ps_Execute := process(manualMode := TRUE, error => error);
END_CASE
END_METHOD

METHOD PRIVATE ps_Holding : BOOL
VAR_INPUT
END_VAR
{warning disable C0371}
//set robot to pause

ps_Holding := TRUE;
END_METHOD

METHOD PRIVATE ps_Resetting : BOOL
VAR_INPUT
END_VAR
{warning disable C0371}
(*reset conveyors*)

ps_Resetting := 
	reset AND
	NOT robotLeft.error AND
	NOT robotRight.error;
END_METHOD

METHOD PRIVATE ps_Starting : BOOL
VAR_INPUT
END_VAR
{warning disable C0371}
//extend conveyors

ps_Starting := TRUE; //conveyors extended
END_METHOD

METHOD PRIVATE ps_Stopping : BOOL
VAR_INPUT
END_VAR
{warning disable C0371}
aoiLoadLeft.reset();
aoiLoadRight.reset();

robotLeft.clearCommand();
robotRight.clearCommand();

//stop conveyors

ps_Stopping :=
	NOT robotLeft.Busy AND
	NOT robotRight.Busy;
END_METHOD

ACTION runPML:
(*
PackML
	state machine for packaging applications - see Tc3_PackML_V2 library on InfoSys
	
	final states - wait for an input or condition and command to new state
	intermediate states - complete a task and call pmlStateMachine.M_StateComplete() to advance to next state
	
the following states currently use the same logic (albeit in different methods), implementation may change later
	ps_Stopping() and ps_Aborting()
	ps_Resetting() and ps_Clearing()
	
STOP - controlled stop **with intent to shutdown or vacate for extended time** induced by operator/HMI - otherwise use HOLD
ABORT - emergency stop due to machine errors


HOLD - minor local issues
SUSPEND - external issues

EXECUTE - major control logic
	different modes may require different tasks
	create methods as required for different modes, then call the correct method in ps_Completing()
	can be commanded to STOP, ABORT, HOLD, or SUSPEND at any point
COMPLETING - process complete, move product out of system and finish transition to COMPLETED
*)

IF //abort at machine error
	robotLeft.error OR 
	robotRight.error
	//+conveyor errors
THEN
	pmlCommand := ePMLCommand_Abort;
	
ELSIF stop THEN //stop at command stop
	pmlCommand := ePMLCommand_Stop;

ELSIF FALSE (*A2.4 cannot allow bundles to enter*) THEN //FALSE condition never executes - this is temporary
	pmlCommand := ePMLCommand_Suspend;
END_IF


CASE pmlState OF
	0: (*ePMLState_Undefined*) //default state on startup
		pmlCommand := ePMLCommand_Stop;
		
	ePMLState_Stopping:
		IF ps_Stopping() THEN
			pmlStateMachine.M_StateComplete();
		END_IF
		
	ePMLState_Stopped:
		pmlCommand := ePMLCommand_Reset;
	
    ePMLState_Resetting:
		IF ps_Resetting() THEN
			reset := FALSE;
			pmlStateMachine.M_StateComplete();
		END_IF
		
	ePMLState_Idle:
		IF execute THEN
			execute := FALSE;
			pmlCommand := ePMLCommand_Start;
		END_IF
	
	ePMLState_Starting:
		IF ps_Starting() THEN
			pmlStateMachine.M_StateComplete();
		END_IF
	
	ePMLState_Execute: 
		IF hold THEN
			pmlCommand := ePMLCommand_Hold;
		END_IF
		IF ps_Execute(error => error) THEN
			pmlStateMachine.M_StateComplete();
			pmlCommand := ePMLCommand_Complete;
		END_IF
		
	ePMLState_Completing:
		pmlStateMachine.M_StateComplete();
	
	ePMLState_Complete:
		pmlCommand := ePMLCommand_Reset;
	
	ePMLState_Holding:
		IF ps_Holding() THEN
			pmlStateMachine.M_StateComplete();
		END_IF
	
	ePMLState_Held:
		IF NOT hold THEN
			pmlCommand := ePMLCommand_Unhold;
		END_IF
	
	ePMLState_Unholding:
		pmlStateMachine.M_StateComplete(); //release all pause commands and IO
	
	ePMLState_Suspended: //based on output section conditions
	ePMLState_Suspending: //based on output section conditions
	ePMLState_Unsuspending: //based on output section conditions
	
	ePMLState_Aborting:
		IF ps_Aborting() THEN
			pmlStateMachine.M_StateComplete();
		END_IF
	
	ePMLState_Aborted:
		pmlCommand := ePMLCommand_Clear;
	
	ePMLState_Clearing:
		IF ps_Clearing() THEN
			pmlStateMachine.M_StateComplete();
		END_IF
	
END_CASE
END_ACTION

END_FUNCTION_BLOCK

// ---- POUs/Utility/AddToArray.TcPOU
FUNCTION AddToArray : BOOL
VAR_INPUT
	arr : POINTER TO BYTE;
	numEntries : LINT;
	dataSize : UDINT;
	
	newEntry : ANY;
END_VAR
VAR
	i : LINT;
END_VAR

//numEntries := (UPPER_BOUND(arr, 1) - LOWER_BOUND(arr, 1) + 1) / dataSize;

FOR i:=0 TO numEntries-1 BY 1 DO
	
	IF ArrayIsEmpty(arr := ADR(arr[i]), arrSize := dataSize) THEN
		AddToArray := MEMCPY(ADR(arr[i]), ADR(newEntry), dataSize) > 0;
		RETURN;
	END_IF
	
END_FOR

END_FUNCTION
